(* CODESYS project NTP145_JIGA03_CPU_NX3030_0001.project
   Version: 3.61.0.0
   Project Profile: Single
   Title: Super Teste NX3030
   Company: Altus S.A.

Project tree, tasks and I/O mapping:
  Device : NX3030, Altus S.A., order no. NX3030, version 1.3.61.200
    application Application
      libraries: NX4000 Diagnostic Structs, 1.0.0.0 (WAA); NJ1001 Diagnostic Structs, 1.0.0.0 (Manufacturer); NJ1005 Diagnostic Structs, 1.0.0.1 (Manufacturer); NJ2001 Diagnostic Structs, 1.0.0.0 (Manufacturer); NJ6000 Diagnostic Structs, 1.0.0.1 (Manufacturer); NJ6001 Diagnostic Structs, 1.0.0.3 (Manufacturer); NJ6005 Diagnostic Structs, 1.0.0.9 (Manufacturer); NJ6010 Diagnostic Structs, 1.0.0.0 (Manufacturer); NJ6011 Diagnostic Structs, 1.0.0.0 (Manufacturer); NJ6020 Diagnostic Structs, 1.0.0.3 (Manufacturer); NJ6100 Diagnostic Structs, 1.0.0.0 (Manufacturer); NJ6101 Diagnostic Structs, 1.0.0.1 (Manufacturer); LibLogs, * (Manufacturer); Util, * (System); NextoSOE, 1.0.0.1 (WAA); LibMQTT, * (Manufacturer); LibRecipeHandler, 1.0.0.2 (Manufacturer); ; RedundancyLib, 3.4.4.31 (3S - Smart Software Solutions GmbH); LibInternal, 1.0.0.15 (Manufacturer); ; NX3030 Diagnostic Structs, 1.1.2.1 (WAA); NX4010 Diagnostic Structs, 1.0.0.3 (WAA); NX5000 Diagnostic Structs, 1.0.0.5 (WAA); NX5001 Diagnostic Structs, 1.0.1.12 (WAA); NXModbus Diagnostic Structs, 1.0.0.5 (WAA); LibRtuStandard, 1.0.0.14 (Manufacturer); IEC 60870-5-104 Server Diagnostic Structs, 1.0.0.2 (Manufacturer); ; ; ; ; 
      task Configuration (cyclic, interval 9000 µs, priority 4) calls Configuration.EtherCAT_Task [Configuration.EtherCAT_Task]
      task MainTask (cyclic, interval 250 ms, priority 13, watchdog 1000 ms x 1) calls MainPrg
      task ATModbusMODBUS_Server_2 (cyclic, interval 60 ms, priority 16) calls MODBUS_Server_2_Instance.Task
      task ATModbusMODBUS_Client_2 (cyclic, interval 41 ms, priority 16) calls MODBUS_Client_2_Instance.Task
      task ATModbusMODBUS_Server_3 (cyclic, interval 20 ms, priority 16) calls MODBUS_Server_3_Instance.Task
      task ATModbusMODBUS_Client_3 (cyclic, interval 41 ms, priority 16) calls MODBUS_Client_3_Instance.Task
      task ATModbusMODBUS_Slave_1 (cyclic, interval 60 ms, priority 16) calls MODBUS_Slave_1_Instance.Task
      task ATModbusMODBUS_Master_1 (cyclic, interval 16 ms, priority 16) calls MODBUS_Master_1_Instance.Task
      Bill of Materials
      Configuration and Consumption
      SystemGVLs/
        global variables System_Diagnostics
        global variables Module_Diagnostics
        global variables IOQualities
        global variables Special_Variables_Redundant
        global variables Special_Variables
      UserGVLs/
        global variables Qualities
        global variables ReqDiagnostics
        global variables Disables
        Non-Redundant/
          global variables ATs
          global variables ProjectConstants
          global variables ModbusSymbol
          global variables NonRedData
          global variables MinMaxTimes
          global variables DiagsRetain
          global variables HwVersions
          global variables Task_Information
          global variables SymbolicsNonRedundant
          global variables NonRedPointer
        Redundant/
          global variables Languages
          global variables PIDs
          global variables QuantityOfVariables
          global variables Symbolics
          global variables Recipe
          global variables ImportExportOnline
          global variables Mask
      SystemPOUs/
        program SpecialVariablesRedundantPrg [ST]
        program SpecialVariablesPrg [ST]
        program MainPrg [ST]
      UserPOUs/
        program StartPrg [ST]
        program NonSkippedPrg [ST]
        program ActivePrg [ST]
        Redundant/
          program CheckLanguages [ST]
          program Alarms [ST]
          program CheckProfibusIOs [ST]
          program PidGenerator [ST]
          program IncrRedData [ST]
          program CheckSoe [ST]
          program StateChange [ST]
          program CheckRecipe [ST]
          program ProfibusStateChange [ST]
          program CheckNVL [ST]
          Languages/
            CFC/
              data type DUT_CFC
              function block FB_CFC [CFC]
              function block FB_CFC_2 [CFC]
              program POU_CFC_1000 [CFC]
            program POU_CFC [CFC]
            program POU_FBD [FBD]
            program POU_IL [IL]
            program POU_LD [LD]
            program POU_SFC [SFC]: Testa_LD_active, Testa_IL_active, Testa_CFC_active, Testa_SFC_active, Testa_FBD_active
          program Recursividade [ST]
          program Iec104Server [ST]: DbpCmdReceiver, StepCmdReceiver
        Non-Redundant/
          program CheckModbus4 [ST]
          program CleanStats [ST]
          program CheckRedData [ST]
          program CheckSntp [ST]
          program UserLog [ST]
          program CycleTimes [ST]
          program CheckModbus1 [ST]
          program CheckModbus3 [ST]
          program CheckModbus2 [ST]
          program CheckDiagsRetain [ST]
          program ReadHwVersions [ST]
          program CheckRam [ST]
          program CheckForcing [ST]
          program WriteHwVersionsNonActive [ST]
          program DaylightSavingTime [ST]
          program MQTT [ST]
          program CheckSpecialVariables [ST]
          program CheckSpecialVarsRed [ST]
      Symbol Configuration
      global variables PersistentVars
      UserFunctions/
        function CONCATENA_2WORD_TO_DWORD [LD]
        function iCounterIncFun [ST]
      UserFunctionsBlocks/
        function block Delay [ST]
        function block Delay1 [ST]
        function block fbTotalizador [CFC]
      UserNVLs/
        global variables NVL_Sender_BroadCast_for_all
        global variables NVL_Sender_JIGA03_Exclusive_to_JIGA01
        global variables NVL_Sender_JIGA03_Exclusive_to_JIGA02
        global variables NVL_Sender_JIGA03_Exclusive_to_JIGA05
        global variables NVL_Sender_JIGA03_Exclusive_to_JIGA07
        declarations NVL_Receiver_JIGA01_Broadcast
        declarations NVL_Receiver_JIGA01_Exclusive
        declarations NVL_Receiver_JIGA02_Broadcast
        declarations NVL_Receiver_JIGA02_Exclusive
        declarations NVL_Receiver_JIGA05_Broadcast
        declarations NVL_Receiver_JIGA05_Exclusive
        declarations NVL_Receiver_JIGA07_Broadcast
        declarations NVL_Receiver_JIGA07_Exclusive
      UserStruct/
        data type Firmware
        data type Firmware_CPU
        data type Task_Informations
        data type NVL_Result
      global variables PidRetainGVL
      program PIDControl [ST]
      RecipeManager
        recipe definition Machine01: Recipe.iRecipeValueA : INT; Recipe.iRecipeValueB : INT; Recipe.iRecipeValueC : INT
      trace Trace (task MainTask): REM05_PO2020_G0, REM05_PO1000_G0, PersistentVars.dwSlave5DigIOsErrors, Task_Information.TI_MainTask.TaskInfo.dwCurScanTime
      Redundancy Configuration
    Configuration : Bus, WAA, order no. Configuration, version 1.1.1.3
      NX3030 : NX3030, Altus S.A., order no. NX3030, version 1.3.61.200
          settings: DC sync0 cycletime = 5000; Cluster Redundancy Enable = True; Generate Error if Task Whatchdog time greater than %80 of interval time = False; Consist retain and persistent area in %Q. = False; Version of MT8500 software.Major = 3; Version of MT8500 software.Minor = 61; Version of MT8500 software.Build = 300; VFInitGenerate = True; Rack Configuration Info.Total Number of Racks = 1; Rack Configuration Info.Rack-0 Type = 9003; IOModule's Address for interrupt = 255; SNTP CONFIGURATION.IP Address of First SNTP Server = [192, 168, 16, 86]; SNTP CONFIGURATION.IP Address = [192, 168, 16, 87]; SOE VARIABLE>.BaseType = 28; SOE VARIABLE>.Address = ADR(PersistentVars.IEC_SOE_QUEUE_INFO); SOE VARIABLE>.SizeInBits = 96096; SOE VARIABLE>.TotalSizeInBits = 96096; Redundancy Without Panel. = FALSE; CurrentProjectProfileParameter = 'Single'; Enable Interface = True; Enable Interface = True
        <Empty>
        COM 1
          MODBUS_Slave_1 : MODBUS RTU Slave, WAA, version 1.0.0.11
              settings: Task Name = 'ATModbusMODBUS_Slave_1'
              unmapped channels: %QD85108 Mapping Disabling
            MODBUS_Slave_1_Mapping_000 : Coil, WAA, version 1.0.0.11
            MODBUS_Slave_1_Mapping_001 : Input Status, WAA, version 1.0.0.11
            MODBUS_Slave_1_Mapping_002 : Holding Register, WAA, version 1.0.0.11
            MODBUS_Slave_1_Mapping_003 : Input Register, WAA, version 1.0.0.11
        COM 2
          MODBUS_Master_1 : MODBUS RTU Master, WAA, version 1.0.0.12
              settings: Task Name = 'ATModbusMODBUS_Master_1'
            MODBUS_Device_11 : MODBUS Device, WAA, version 1.0.0.12
                unmapped channels: %QD85132 Mapping Disabling
              MODBUS_Device_11_Mapping_000 : Coil, WAA, version 1.0.0.12
              MODBUS_Device_11_Mapping_001 : Input Status, WAA, version 1.0.0.12
              MODBUS_Device_11_Mapping_002 : Holding Register, WAA, version 1.0.0.12
              MODBUS_Device_11_Mapping_003 : Input Register, WAA, version 1.0.0.12
              MODBUS_Device_11_Mapping_004 : Coil, WAA, version 1.0.0.12
              MODBUS_Device_11_Mapping_005 : Holding Register, WAA, version 1.0.0.12
        NET 1
            settings: IP Address = [192, 168, 23, 0]; Subnetwork Mask = [255, 255, 248, 0]; Gateway Address = [192, 168, 16, 253]; IP Address PLC A Non Active = [192, 168, 23, 1]; IP Address PLC B Non Active = [192, 168, 23, 2]; Redundant = TRUE; IP Address PLC B Active = [192, 168, 23, 0]; Enable Interface = True; Switchover in case of Ethernet failure = TRUE; Obtain an IP address automatically (Single Mode) = False
          MODBUS_Client_4 : MODBUS Symbol Client, Altus S.A., version 1.0.0.37
              settings: Diagnostic Variable.BaseType = 28; Diagnostic Variable.Address = ADR(System_Diagnostics.DG_MODBUS_Client_4); Diagnostic Variable.SizeInBits = 160; Diagnostic Variable.TotalSizeInBits = 160
            MODBUS_Device_41 : MODBUS Device, Altus S.A., version 1.0.0.37
                settings: IP Address = [192, 168, 23, 3]; Mappings definition.Count = 6; Item_00000.Value Variable.BaseType = 3; Item_00000.Value Variable.Address = ADR(ModbusSymbol.awModbus4HoldingWrite); Item_00000.Value Variable.SizeInBits = 16; Item_00000.Value Variable.TotalSizeInBits = 1920; Item_00001.Value Variable.BaseType = 3; Item_00001.Value Variable.Address = ADR(ModbusSymbol.awModbus4HoldingRead); Item_00001.Value Variable.SizeInBits = 16; Item_00001.Value Variable.TotalSizeInBits = 1920; Item_00002.Value Variable.BaseType = 0; Item_00002.Value Variable.Address = ADR(ModbusSymbol.abModbus4CoilsWrite); Item_00002.Value Variable.SizeInBits = 8; Item_00002.Value Variable.TotalSizeInBits = 15360; Item_00003.Value Variable.BaseType = 0; Item_00003.Value Variable.Address = ADR(ModbusSymbol.abModbus4CoilsRead); Item_00003.Value Variable.SizeInBits = 8; Item_00003.Value Variable.TotalSizeInBits = 15360; Item_00004.Value Variable.BaseType = 3; Item_00004.Value Variable.Address = ADR(ModbusSymbol.awModbus4InputRegRead); Item_00004.Value Variable.SizeInBits = 16; Item_00004.Value Variable.TotalSizeInBits = 1920; Item_00005.Value Variable.BaseType = 0; Item_00005.Value Variable.Address = ADR(ModbusSymbol.abModbus4StatusRead); Item_00005.Value Variable.SizeInBits = 8; Item_00005.Value Variable.TotalSizeInBits = 15360; Requests definition.Count = 6; Item_00000.Diagnostic Variable.BaseType = 28; Item_00000.Diagnostic Variable.Address = ADR(ReqDiagnostics.MODBUS_Device_41_REQDG_0001); Item_00000.Diagnostic Variable.SizeInBits = 64; Item_00000.Diagnostic Variable.TotalSizeInBits = 64; Item_00000.Disabling Variable.BaseType = 0; Item_00000.Disabling Variable.Address = ADR(Disables.MODBUS_Device_41_DISABLE_0001); Item_00000.Disabling Variable.SizeInBits = 8; Item_00000.Disabling Variable.TotalSizeInBits = 8; Item_00001.Diagnostic Variable.BaseType = 28; Item_00001.Diagnostic Variable.Address = ADR(ReqDiagnostics.MODBUS_Device_41_REQDG_0002); Item_00001.Diagnostic Variable.SizeInBits = 64; Item_00001.Diagnostic Variable.TotalSizeInBits = 64; Item_00001.Disabling Variable.BaseType = 0;
                  Item_00001.Disabling Variable.Address = ADR(Disables.MODBUS_Device_41_DISABLE_0002); Item_00001.Disabling Variable.SizeInBits = 8; Item_00001.Disabling Variable.TotalSizeInBits = 8; Item_00002.Diagnostic Variable.BaseType = 28; Item_00002.Diagnostic Variable.Address = ADR(ReqDiagnostics.MODBUS_Device_41_REQDG_0003); Item_00002.Diagnostic Variable.SizeInBits = 64; Item_00002.Diagnostic Variable.TotalSizeInBits = 64; Item_00002.Disabling Variable.BaseType = 0; Item_00002.Disabling Variable.Address = ADR(Disables.MODBUS_Device_41_DISABLE_0003); Item_00002.Disabling Variable.SizeInBits = 8; Item_00002.Disabling Variable.TotalSizeInBits = 8; Item_00003.Diagnostic Variable.BaseType = 28; Item_00003.Diagnostic Variable.Address = ADR(ReqDiagnostics.MODBUS_Device_41_REQDG_0004); Item_00003.Diagnostic Variable.SizeInBits = 64; Item_00003.Diagnostic Variable.TotalSizeInBits = 64; Item_00003.Disabling Variable.BaseType = 0; Item_00003.Disabling Variable.Address = ADR(Disables.MODBUS_Device_41_DISABLE_0004); Item_00003.Disabling Variable.SizeInBits = 8; Item_00003.Disabling Variable.TotalSizeInBits = 8; Item_00004.Diagnostic Variable.BaseType = 28; Item_00004.Diagnostic Variable.Address = ADR(ReqDiagnostics.MODBUS_Device_41_REQDG_0005); Item_00004.Diagnostic Variable.SizeInBits = 64; Item_00004.Diagnostic Variable.TotalSizeInBits = 64; Item_00004.Disabling Variable.BaseType = 0; Item_00004.Disabling Variable.Address = ADR(Disables.MODBUS_Device_41_DISABLE_0005); Item_00004.Disabling Variable.SizeInBits = 8; Item_00004.Disabling Variable.TotalSizeInBits = 8; Item_00005.Diagnostic Variable.BaseType = 28; Item_00005.Diagnostic Variable.Address = ADR(ReqDiagnostics.MODBUS_Device_41_REQDG_0006); Item_00005.Diagnostic Variable.SizeInBits = 64; Item_00005.Diagnostic Variable.TotalSizeInBits = 64; Item_00005.Disabling Variable.BaseType = 0; Item_00005.Disabling Variable.Address = ADR(Disables.MODBUS_Device_41_DISABLE_0006); Item_00005.Disabling Variable.SizeInBits = 8; Item_00005.Disabling Variable.TotalSizeInBits = 8
          MODBUS_Server_2 : MODBUS Server, WAA, version 1.0.0.13
              settings: Task Name = 'ATModbusMODBUS_Server_2'
              unmapped channels: %QD85164 Mapping Disabling
            MODBUS_Server_2_Mapping_000 : Holding Register, WAA, version 1.0.0.13
                settings: Write Filter IP = [192, 168, 23, 3]; Write Filter Mask = [255, 255, 255, 255]; Read Filter IP = [192, 168, 23, 3]; Read Filter Mask = [255, 255, 255, 255]
            MODBUS_Server_2_Mapping_001 : Coil, WAA, version 1.0.0.13
                settings: Write Filter IP = [192, 168, 23, 3]; Write Filter Mask = [255, 255, 255, 255]; Read Filter IP = [192, 168, 23, 3]; Read Filter Mask = [255, 255, 255, 255]
            MODBUS_Server_2_Mapping_002 : Input Register, WAA, version 1.0.0.13
                settings: Read Filter IP = [192, 168, 23, 3]; Read Filter Mask = [255, 255, 255, 255]
            MODBUS_Server_2_Mapping_003 : Input Status, WAA, version 1.0.0.13
                settings: Read Filter IP = [192, 168, 23, 3]; Read Filter Mask = [255, 255, 255, 255]
          IEC_104_Server : IEC 60870-5-104 Server, Altus S.A., version 1.0.0.21
              settings: Diagnostic Variable.BaseType = 28; Diagnostic Variable.Address = ADR(Module_Diagnostics.DG_IEC_104_Server); Diagnostic Variable.SizeInBits = 1472; Diagnostic Variable.TotalSizeInBits = 1472
            JIGA11_CPU_HX3040_Client : Client, Altus S.A., version 1.0.0.21
                settings: Parameter list definition.Count = 15; Item_00000.Value Variable.BaseType = 0; Item_00000.Value Variable.Address = ADR(Iec104Server.bDI); Item_00000.Value Variable.SizeInBits = 8; Item_00000.Value Variable.TotalSizeInBits = 8; Item_00001.Value Variable.BaseType = 0; Item_00001.Value Variable.Address = ADR(Iec104Server.bDO); Item_00001.Value Variable.SizeInBits = 8; Item_00001.Value Variable.TotalSizeInBits = 8; Item_00002.Value Variable.BaseType = 28; Item_00002.Value Variable.Address = ADR(Iec104Server.dbpI); Item_00002.Value Variable.SizeInBits = 16; Item_00002.Value Variable.TotalSizeInBits = 16; Item_00003.Value Variable.BaseType = 28; Item_00003.Value Variable.Address = ADR(Iec104Server.dbpO); Item_00003.Value Variable.SizeInBits = 16; Item_00003.Value Variable.TotalSizeInBits = 16; Item_00004.Value Variable.BaseType = 10; Item_00004.Value Variable.Address = ADR(Iec104Server.usiSP); Item_00004.Value Variable.SizeInBits = 8; Item_00004.Value Variable.TotalSizeInBits = 8; Item_00005.Value Variable.BaseType = 28; Item_00005.Value Variable.Address = ADR(Iec104Server.dbpStep); Item_00005.Value Variable.SizeInBits = 16; Item_00005.Value Variable.TotalSizeInBits = 16; Item_00006.Value Variable.BaseType = 7; Item_00006.Value Variable.Address = ADR(Iec104Server.iAIn); Item_00006.Value Variable.SizeInBits = 16; Item_00006.Value Variable.TotalSizeInBits = 16; Item_00007.Value Variable.BaseType = 7; Item_00007.Value Variable.Address = ADR(Iec104Server.iAOn); Item_00007.Value Variable.SizeInBits = 16; Item_00007.Value Variable.TotalSizeInBits = 16; Item_00008.Value Variable.BaseType = 7; Item_00008.Value Variable.Address = ADR(Iec104Server.iAIs); Item_00008.Value Variable.SizeInBits = 16; Item_00008.Value Variable.TotalSizeInBits = 16; Item_00009.Value Variable.BaseType = 7; Item_00009.Value Variable.Address = ADR(Iec104Server.iAOs); Item_00009.Value Variable.SizeInBits = 16;
                  Item_00009.Value Variable.TotalSizeInBits = 16; Item_00010.Value Variable.BaseType = 14; Item_00010.Value Variable.Address = ADR(Iec104Server.rAIf); Item_00010.Value Variable.SizeInBits = 32; Item_00010.Value Variable.TotalSizeInBits = 32; Item_00011.Value Variable.BaseType = 14; Item_00011.Value Variable.Address = ADR(Iec104Server.rAOf); Item_00011.Value Variable.SizeInBits = 32; Item_00011.Value Variable.TotalSizeInBits = 32; Item_00012.Value Variable.BaseType = 8; Item_00012.Value Variable.Address = ADR(Iec104Server.diIT); Item_00012.Value Variable.SizeInBits = 32; Item_00012.Value Variable.TotalSizeInBits = 32; Item_00012.Counter Variable.BaseType = 8; Item_00012.Counter Variable.Address = ADR(IEC104Server.diITCounter); Item_00012.Counter Variable.SizeInBits = 32; Item_00012.Counter Variable.TotalSizeInBits = 32; Item_00013.Value Variable.BaseType = 10; Item_00013.Value Variable.Address = ADR(Iec104Server.usiJigId); Item_00013.Value Variable.SizeInBits = 8; Item_00013.Value Variable.TotalSizeInBits = 8; Item_00014.Value Variable.BaseType = 10; Item_00014.Value Variable.Address = ADR(Iec104Server.usiJigId); Item_00014.Value Variable.SizeInBits = 8; Item_00014.Value Variable.TotalSizeInBits = 8
        NET 2
            settings: IP Address = [192, 168, 23, 0]; Subnetwork Mask = [255, 255, 248, 0]; IP Address PLC A Non Active = [192, 168, 23, 1]; IP Address PLC B Non Active = [192, 168, 23, 2]; IP Address PLC B Active = [192, 168, 23, 0]; Enable Interface = True; Switchover in case of Ethernet failure = TRUE
        NX8000 : NX8000, Altus S.A., order no. NX8000, version 1.3.61.200
            settings: DC sync0 cycletime = 5000; Diag Instance Id = 0
        NX4010 : NX4010, Altus S.A., order no. NX4010, version 1.3.61.200
            settings: Physical Address of the Slave = 4; DC sync0 cycletime = 5000; Diag Instance Id = 4; %Q Start Address of Diagnostics Area = 82634; Input Offset = 81920; Output Offset = 81920
            unmapped channels: %QB81920 Reserved, %IW81920 Reserved
        NX5001_2 : NX5001, Altus S.A., order no. NX5001, version 1.1.1.19
            settings: Physical Address of the Slave = 8; Diag Instance Id = 8; %Q Start Address of Module Diagnostics Area = 83000; %Q Start Address of Slaves Diagnostics Area = 65536; User Commands Offset = 81921; NX5001R = 1; Fast Diagnostics Offset = 81924; DpParameter.Station address = 1; UseDefaults = FALSE
            unmapped channels: %QB81921 User Commands, %IW81924 User Status
        NX5001_3 : NX5001, Altus S.A., order no. NX5001, version 1.1.1.19
            settings: Physical Address of the Slave = 16; Diag Instance Id = 16; %Q Start Address of Module Diagnostics Area = 83086; %Q Start Address of Slaves Diagnostics Area = 65717; User Commands Offset = 81923; Identification = 2; Fast Diagnostics Offset = 81928; Manual user change the %Q Start Address of Slaves = TRUE; SlaveMaxDiagDataLen.Slave0 = 25; DpParameter.Station address = 1
            unmapped channels: %QB81923 User Commands, %IW81928 User Status
          PO5063_04 : PO5063, Altus S.A., order no. PO5063, version Revision=1.30, HW=V100, SW=5.00
              settings: SlavePrmData.wdFact1 = 1; SlavePrmData.wdFact2 = 100; SlavePrmData.userPrmData.userParameter = [0,4,35,0,20]; StationAddress = 4
            REM04_PO1000 : PO1000 16DI 24 Vdc Opto Coupled , Altus S.A., order no. PO1000, version Revision=1.30, HW=V100, SW=5.00
                input  REM04_PO1000_G0 : BYTE  // Input0.Byte0
                input  REM04_PO1000_G1 : BYTE  // Input0.Byte1
                unmapped channels: %IB24 Input0
        NX5000_1 : NX5000, Altus S.A., order no. NX5000, version 1.3.61.200
            settings: Physical Address of the Slave = 10; DC sync0 cycletime = 5000; Diag Instance Id = 10; %Q Start Address of Module Diagnostics Area = 83344; Network Redundancy = 1; User Commands Offset = 81929; Fast Diagnostics Offset = 81940; Enable Interface = True
            unmapped channels: %QB81929 Reserved, %IW81940 Reserved
          NET 1
              settings: IP Address = [192, 168, 23, 3]; Subnetwork Mask = [255, 255, 248, 0]; Gateway Address = [192, 168, 16, 253]; IP Address PLC A Non Active = [192, 168, 23, 4]; IP Address PLC B Non Active = [192, 168, 23, 5]; Redundant = TRUE; IP Address PLC B Active = [192, 168, 23, 3]; Enable Interface = True
            MODBUS_Server_4 : MODBUS Symbol Server, Altus S.A., version 1.0.0.8
                settings: Write Filter IP Address = [192, 168, 23, 0]; Write Filter Mask = [255, 255, 255, 248]; Read Filter IP Address = [192, 168, 23, 0]; Read Filter Mask = [255, 255, 255, 248]; Parameter list definition.Count = 4; Item_00000.Value Variable.BaseType = 3; Item_00000.Value Variable.Address = ADR(ModbusSymbol.awModbus4Holding); Item_00000.Value Variable.SizeInBits = 16; Item_00000.Value Variable.TotalSizeInBits = 1920; Item_00001.Value Variable.BaseType = 0; Item_00001.Value Variable.Address = ADR(ModbusSymbol.abModbus4Coils); Item_00001.Value Variable.SizeInBits = 8; Item_00001.Value Variable.TotalSizeInBits = 15360; Item_00002.Value Variable.BaseType = 3; Item_00002.Value Variable.Address = ADR(ModbusSymbol.awModbus4InputReg); Item_00002.Value Variable.SizeInBits = 16; Item_00002.Value Variable.TotalSizeInBits = 1920; Item_00003.Value Variable.BaseType = 0; Item_00003.Value Variable.Address = ADR(ModbusSymbol.abModbus4Status); Item_00003.Value Variable.SizeInBits = 8; Item_00003.Value Variable.TotalSizeInBits = 15360; Diagnostic Variable.BaseType = 28; Diagnostic Variable.Address = ADR(Module_Diagnostics.DG_MODBUS_Server_4); Diagnostic Variable.SizeInBits = 160; Diagnostic Variable.TotalSizeInBits = 160
            MODBUS_Client_2 : MODBUS Client, WAA, version 1.0.0.14
                settings: Task Name = 'ATModbusMODBUS_Client_2'
              MODBUS_Device_21 : MODBUS Device, WAA, version 1.0.0.14
                  settings: Destination IP = [192, 168, 23, 0]
                  unmapped channels: %QD85020 Mapping Disabling
                MODBUS_Device_21_Mapping_001 : Holding Register, WAA, version 1.0.0.14
                MODBUS_Device_21_Mapping_002 : Holding Register, WAA, version 1.0.0.14
                MODBUS_Device_21_Mapping_003 : Coil, WAA, version 1.0.0.14
                MODBUS_Device_21_Mapping_004 : Coil, WAA, version 1.0.0.14
                MODBUS_Device_21_Mapping_005 : Input Register, WAA, version 1.0.0.14
                MODBUS_Device_21_Mapping_006 : Input Status, WAA, version 1.0.0.14
            MODBUS_Server_3 : MODBUS Server, WAA, version 1.0.0.13
                settings: Task Name = 'ATModbusMODBUS_Server_3'
                unmapped channels: %QD85052 Mapping Disabling
              MODBUS_Server_3_Mapping_001 : Holding Register, WAA, version 1.0.0.13
                  settings: Write Filter IP = [192, 168, 23, 6]; Write Filter Mask = [255, 255, 255, 255]; Read Filter IP = [192, 168, 23, 6]; Read Filter Mask = [255, 255, 255, 255]
              MODBUS_Server_3_Mapping_002 : Coil, WAA, version 1.0.0.13
                  settings: Write Filter IP = [192, 168, 23, 6]; Write Filter Mask = [255, 255, 255, 255]; Read Filter IP = [192, 168, 23, 6]; Read Filter Mask = [255, 255, 255, 255]
              MODBUS_Server_3_Mapping_003 : Input Register, WAA, version 1.0.0.13
                  settings: Read Filter IP = [192, 168, 23, 6]; Read Filter Mask = [255, 255, 255, 255]
              MODBUS_Server_3_Mapping_004 : Input Status, WAA, version 1.0.0.13
                  settings: Read Filter IP = [192, 168, 23, 6]; Read Filter Mask = [255, 255, 255, 255]
        NX5000_2 : NX5000, Altus S.A., order no. NX5000, version 1.3.61.200
            settings: Physical Address of the Slave = 12; DC sync0 cycletime = 5000; Diag Instance Id = 12; %Q Start Address of Module Diagnostics Area = 83544; User Commands Offset = 81931; NX5000R = 1; Fast Diagnostics Offset = 81946; Enable Interface = True
            unmapped channels: %QB81931 Reserved, %IW81946 Reserved
          NET 1
              settings: IP Address = [192, 168, 23, 3]; Subnetwork Mask = [255, 255, 248, 0]; Gateway Address = [192, 168, 16, 253]; IP Address PLC A Non Active = [192, 168, 23, 4]; IP Address PLC B Non Active = [192, 168, 23, 5]; IP Address PLC B Active = [192, 168, 23, 3]; Enable Interface = True
        NX5001_1 : NX5001, Altus S.A., order no. NX5001, version 1.1.1.19
            settings: Physical Address of the Slave = 6; Diag Instance Id = 6; %Q Start Address of Module Diagnostics Area = 83172; %Q Start Address of Slaves Diagnostics Area = 65536; Network Redundancy = 1; User Commands Offset = 81925; Fast Diagnostics Offset = 81932; Manual user change the %Q Start Address of Slaves = TRUE; SlaveMaxDiagDataLen.Slave0 = 25; SlaveMaxDiagDataLen.Slave1 = 25; DpParameter.Station address = 1; UseDefaults = FALSE
            unmapped channels: %QB81925 User Commands, %IW81932 User Status
          PO5065_05 : PO5065, Altus S.A., order no. PO5065, version Revision=1.30, HW=V100, SW=1.01
              settings: SlavePrmData.wdFact1 = 1; SlavePrmData.wdFact2 = 100; SlavePrmData.userPrmData.userParameter = [0, 0, 0, 0, 4, 98, 0, 20]; StationAddress = 5
            REM05_PO1000 : PO1000 16DI 24 Vdc Opto Coupled , Altus S.A., order no. PO1000, version Revision=1.30, HW=V100, SW=1.01
                input  REM05_PO1000_G0 : BYTE  // Input0.Byte0
                input  REM05_PO1000_G1 : BYTE  // Input0.Byte1
                unmapped channels: %IB0 Input0
            REM05_PO2020 : PO2020 16DO Transistor Opto     , Altus S.A., order no. PO2020, version Revision=1.30, HW=V100, SW=1.01
                output REM05_PO2020_G0 : BYTE  // Output0.Byte0
                output REM05_PO2020_G1 : BYTE  // Output0.Byte1
                unmapped channels: %QB2000 Output0
            REM05_PO9100 : PO9100 - Redundant Head PO5065  , Altus S.A., order no. PO9100_RH, version Revision=1.30, HW=V100, SW=1.01
                input  REM05_PO5065_IN AT %IW2 : WORD  // Input0
                output REM05_PO5065_OUT AT %QW2002 : WORD  // Output0
          PO5065_10 : PO5065, Altus S.A., order no. PO5065, version Revision=1.30, HW=V100, SW=1.01
              settings: SlavePrmData.wdFact1 = 1; SlavePrmData.wdFact2 = 100; SlavePrmData.userPrmData.userParameter = [0, 0, 0, 0, 4, 98, 0, 20]; StationAddress = 10
            REM10_PO1212 : PO1212 8AI Universal Isolated   , Altus S.A., order no. PO1212, version Revision=1.30, HW=V100, SW=1.01
                settings: ExtPrmData.userParameter = [10, 8, 10, 4, 4, 4, 4, 4, 4, 4]
                input  REM10_PO1212_C00 : WORD  // Input0.Word0
                input  REM10_PO1212_C01 : WORD  // Input0.Word1
                input  REM10_PO1212_C02 : WORD  // Input0.Word2
                input  REM10_PO1212_C03 : WORD  // Input0.Word3
                input  REM10_PO1212_C04 : WORD  // Input0.Word4
                input  REM10_PO1212_C05 : WORD  // Input0.Word5
                input  REM10_PO1212_C06 : WORD  // Input0.Word6
                input  REM10_PO1212_C07 : WORD  // Input0.Word7
                unmapped channels: %IW4 Input0
            REM10_PO2132 : PO2132 4AO Universal Isolated   , Altus S.A., order no. PO2132, version Revision=1.30, HW=V100, SW=1.01
                settings: ExtPrmData.userParameter = [6, 0, 0, 2, 2, 2]
                output REM10_PO2132_C00 : WORD  // Output0.Word0
                output REM10_PO2132_C01 : WORD  // Output0.Word1
                output REM10_PO2132_C02 : WORD  // Output0.Word2
                output REM10_PO2132_C03 : WORD  // Output0.Word3
                unmapped channels: %QW2004 Output0
            REM10_PO9100 : PO9100 - Redundant Head PO5065  , Altus S.A., order no. PO9100_RH, version Revision=1.30, HW=V100, SW=1.01
                input  REM10_PO5065_IN AT %IW20 : WORD  // Input0
                output REM10_PO5065_OUT AT %QW2012 : WORD  // Output0
        NX5000_3 : NX5000, Altus S.A., order no. NX5000, version 1.3.61.200
            settings: Physical Address of the Slave = 20; DC sync0 cycletime = 5000; Diag Instance Id = 20; %Q Start Address of Module Diagnostics Area = 83744; User Commands Offset = 81933; Fast Diagnostics Offset = 81952; Enable Interface = True
            unmapped channels: %QB81933 Reserved, %IW81952 Reserved
          NET 1
              settings: IP Address = [192, 168, 23, 6]; Subnetwork Mask = [255, 255, 248, 0]; Gateway Address = [192, 168, 16, 253]; IP Address PLC A Non Active = [192, 168, 23, 7]; IP Address PLC B Non Active = [192, 168, 23, 8]; IP Address PLC B Active = [192, 168, 23, 6]; Enable Interface = True
            MODBUS_Client_3 : MODBUS Client, WAA, version 1.0.0.14
                settings: Task Name = 'ATModbusMODBUS_Client_3'
              MODBUS_Device_31 : MODBUS Device, WAA, version 1.0.0.14
                  settings: Destination IP = [192, 168, 23, 3]
                  unmapped channels: %QD85076 Mapping Disabling
                MODBUS_Device_31_Mapping_000 : Holding Register, WAA, version 1.0.0.14
                MODBUS_Device_31_Mapping_001 : Holding Register, WAA, version 1.0.0.14
                MODBUS_Device_31_Mapping_002 : Coil, WAA, version 1.0.0.14
                MODBUS_Device_31_Mapping_003 : Coil, WAA, version 1.0.0.14
                MODBUS_Device_31_Mapping_004 : Input Register, WAA, version 1.0.0.14
                MODBUS_Device_31_Mapping_005 : Input Status, WAA, version 1.0.0.14
  Library Information/
    function GetLibVersion [ST]
    function GetLibVersionNumber [ST]
    function IsLibReleased [ST]
  Project Information/
    function GetCompany [ST]
    function GetTitle [ST]
    function GetVersion [ST]
    function GetTextProperty [ST]
    function GetTextProperty2 [ST]
    function GetNumberProperty [ST]
    function GetBooleanProperty [ST]
    function GetVersionProperty [ST]
  function ForceScanTime [ST]
*)

// Device/Application/UserPOUs/Redundant/Languages/CFC/DUT_CFC
TYPE DUT_CFC :
STRUCT
	iVar01_Add_A: INT;
	iVar02_Add_B: INT;
END_STRUCT
END_TYPE

// Device/Application/UserStruct/Firmware
TYPE Firmware :
STRUCT
	dwFirmwareVersion:	DWORD; // Versão Firmware do produto em Hexadecimal
	uiSlaveAddress: 	UINT; // Rack e Slot do produto em Hexadecimal
	dwProductID:		DWORD; // Modelo do produto em Hexadecimal
	iIndex:				INT; // Ponteiro do local das informações lidas do NextoBus.
END_STRUCT
END_TYPE

// Device/Application/UserStruct/Firmware_CPU
TYPE Firmware_CPU :
STRUCT
	abyCPUVersion: ARRAY[0..3] OF BYTE;		   // Versão da CPU
	abyBootloaderVersion: ARRAY[0..3] OF BYTE; // Versão da CPU
	abyProcAuxVersion: ARRAY[0..3] OF BYTE;	   // Versão da CPU
	dwCPUModel: DWORD;                         // Modelo da CPU
END_STRUCT
END_TYPE

// Device/Application/UserStruct/Task_Informations
TYPE Task_Informations :
STRUCT
	sTaskName:			STRING;						// Variável recebe o nome da tarefa.
	psTaskName:			POINTER TO STRING;			// Ponteiro com o nome da tarefa.
	pstTaskInfo:		POINTER TO stTaskInfo;		// Ponteiro que irá receber as informações da tarefa.
	TaskInfo:			stTaskInfo;					// Retona aqui as Informações sobre a tarefa
END_STRUCT
END_TYPE

// Device/Application/UserStruct/NVL_Result
TYPE NVL_Result :
STRUCT
	iTempoMinimo 				:	INT;	// Tempo do menor intervalo de comunicação
	iTempoMedio					:	INT;	// Tempo médio de intervalo de comunicação
	iTempoMaximo				:	INT;	// Tempo do maior intervalo de comunicação (limite 30000)
	lwQtdTotalComunicacoes		:	LWORD;	// Quantidade total de comunicações realizadas
	wQtdComMaior3segundos		: 	WORD;	//Quantidde de comunicações acima de 3 segundos
	wQtdComMaior4segundos		: 	WORD;	//Quantidde de comunicações acima de 3 segundos
	wQtdComMaior5segundos		: 	WORD;	//Quantidde de comunicações acima de 3 segundos
END_STRUCT
END_TYPE

// Device/Application/SystemGVLs/System_Diagnostics
VAR_GLOBAL
	//DG_MODBUS_Client_4 diagnostics variable
	DG_MODBUS_Client_4                          : T_DIAG_MODBUS_ETH_CLIENT_1;
	//DG_PO5065_05 diagnostics variable
	DG_PO5065_05                    AT %QB65536 : T_DIAG_PO5065_1;
	//DG_REM05_PO1000 diagnostics variable
	DG_REM05_PO1000                 AT %QB65561 : T_DIAG_PO1000_1;
	//DG_REM05_PO2020 diagnostics variable
	DG_REM05_PO2020                 AT %QB65571 : T_DIAG_PO2020_1;
	//DG_REM05_PO9100 diagnostics variable
	DG_REM05_PO9100                 AT %QB65581 : T_DIAG_VIRTUAL_MODULE_1;
	//DG_PO5065_10 diagnostics variable
	DG_PO5065_10                    AT %QB65591 : T_DIAG_PO5065_1;
	//DG_REM10_PO1212 diagnostics variable
	DG_REM10_PO1212                 AT %QB65616 : T_DIAG_PO1212_1;
	//DG_REM10_PO2132 diagnostics variable
	DG_REM10_PO2132                 AT %QB65626 : T_DIAG_PO2134_1;
	//DG_REM10_PO9100 diagnostics variable
	DG_REM10_PO9100                 AT %QB65636 : T_DIAG_VIRTUAL_MODULE_1;
	//DG_PO5063_04 diagnostics variable
	DG_PO5063_04                    AT %QB65717 : T_DIAG_PO5063_1;
	//DG_REM04_PO1000 diagnostics variable
	DG_REM04_PO1000                 AT %QB65742 : T_DIAG_PO1000_1;
	//DG_NX3030 diagnostics variable
	DG_NX3030                       AT %QB81941 : T_DIAG_NX3030_1;
	//DG_MODBUS_Client_2 diagnostics variable
	DG_MODBUS_Client_2              AT %QB85000 : T_DIAG_MODBUS_ETH_CLIENT_1;
	//DG_MODBUS_Device_21_Mapping_001 diagnostics variable
	DG_MODBUS_Device_21_Mapping_001 AT %QB85024 : T_DIAG_MODBUS_ETH_MAPPING_1;
	//DG_MODBUS_Client_3 diagnostics variable
	DG_MODBUS_Client_3              AT %QB85056 : T_DIAG_MODBUS_ETH_CLIENT_1;
	//DG_MODBUS_Device_31_Mapping_000 diagnostics variable
	DG_MODBUS_Device_31_Mapping_000 AT %QB85080 : T_DIAG_MODBUS_ETH_MAPPING_1;
	//DG_MODBUS_Master_1 diagnostics variable
	DG_MODBUS_Master_1              AT %QB85112 : T_DIAG_MODBUS_RTU_MASTER_1;
	//DG_MODBUS_Device_11_Mapping_000 diagnostics variable
	DG_MODBUS_Device_11_Mapping_000 AT %QB85136 : T_DIAG_MODBUS_RTU_MAPPING_1;
	//DG_MODBUS_Device_11_Mapping_001 diagnostics variable
	DG_MODBUS_Device_11_Mapping_001 AT %QB85168 : T_DIAG_MODBUS_RTU_MAPPING_1;
	//DG_MODBUS_Device_11_Mapping_002 diagnostics variable
	DG_MODBUS_Device_11_Mapping_002 AT %QB85176 : T_DIAG_MODBUS_RTU_MAPPING_1;
	//DG_MODBUS_Device_11_Mapping_003 diagnostics variable
	DG_MODBUS_Device_11_Mapping_003 AT %QB85184 : T_DIAG_MODBUS_RTU_MAPPING_1;
	//DG_MODBUS_Device_11_Mapping_004 diagnostics variable
	DG_MODBUS_Device_11_Mapping_004 AT %QB85192 : T_DIAG_MODBUS_RTU_MAPPING_1;
	//DG_MODBUS_Device_11_Mapping_005 diagnostics variable
	DG_MODBUS_Device_11_Mapping_005 AT %QB85200 : T_DIAG_MODBUS_RTU_MAPPING_1;
	//DG_MODBUS_Device_31_Mapping_001 diagnostics variable
	DG_MODBUS_Device_31_Mapping_001 AT %QB85208 : T_DIAG_MODBUS_ETH_MAPPING_1;
	//DG_MODBUS_Device_31_Mapping_002 diagnostics variable
	DG_MODBUS_Device_31_Mapping_002 AT %QB85216 : T_DIAG_MODBUS_ETH_MAPPING_1;
	//DG_MODBUS_Device_31_Mapping_003 diagnostics variable
	DG_MODBUS_Device_31_Mapping_003 AT %QB85224 : T_DIAG_MODBUS_ETH_MAPPING_1;
	//DG_MODBUS_Device_31_Mapping_004 diagnostics variable
	DG_MODBUS_Device_31_Mapping_004 AT %QB85232 : T_DIAG_MODBUS_ETH_MAPPING_1;
	//DG_MODBUS_Device_31_Mapping_005 diagnostics variable
	DG_MODBUS_Device_31_Mapping_005 AT %QB85240 : T_DIAG_MODBUS_ETH_MAPPING_1;
	//DG_MODBUS_Device_21_Mapping_002 diagnostics variable
	DG_MODBUS_Device_21_Mapping_002 AT %QB85248 : T_DIAG_MODBUS_ETH_MAPPING_1;
	//DG_MODBUS_Device_21_Mapping_003 diagnostics variable
	DG_MODBUS_Device_21_Mapping_003 AT %QB85256 : T_DIAG_MODBUS_ETH_MAPPING_1;
	//DG_MODBUS_Device_21_Mapping_004 diagnostics variable
	DG_MODBUS_Device_21_Mapping_004 AT %QB85264 : T_DIAG_MODBUS_ETH_MAPPING_1;
	//DG_MODBUS_Device_21_Mapping_005 diagnostics variable
	DG_MODBUS_Device_21_Mapping_005 AT %QB85272 : T_DIAG_MODBUS_ETH_MAPPING_1;
	//DG_MODBUS_Device_21_Mapping_006 diagnostics variable
	DG_MODBUS_Device_21_Mapping_006 AT %QB85280 : T_DIAG_MODBUS_ETH_MAPPING_1;
END_VAR

// Device/Application/SystemGVLs/Module_Diagnostics
VAR_GLOBAL
	//DG_IEC_104_Server diagnostics variable
	DG_IEC_104_Server              : T_DIAG_IEC104_SERVER_1;
	//DG_MODBUS_Server_4 diagnostics variable
	DG_MODBUS_Server_4             : T_DIAG_MODBUS_ETH_SERVER_1;
	//DG_NX4010 diagnostics variable
	DG_NX4010          AT %QB82634 : T_DIAG_NX4010_1;
	//DG_NX5001_2 diagnostics variable
	DG_NX5001_2        AT %QB83000 : T_DIAG_NX5001_1;
	//DG_NX5001_3 diagnostics variable
	DG_NX5001_3        AT %QB83086 : T_DIAG_NX5001_1;
	//DG_NX5001_1 diagnostics variable
	DG_NX5001_1        AT %QB83172 : T_DIAG_NX5001_1;
	//DG_NX5000_1 diagnostics variable
	DG_NX5000_1        AT %QB83344 : T_DIAG_NX5000_1;
	//DG_NX5000_2 diagnostics variable
	DG_NX5000_2        AT %QB83544 : T_DIAG_NX5000_1;
	//DG_NX5000_3 diagnostics variable
	DG_NX5000_3        AT %QB83744 : T_DIAG_NX5000_1;
	//DG_MODBUS_Server_3 diagnostics variable
	DG_MODBUS_Server_3 AT %QB85032 : T_DIAG_MODBUS_ETH_SERVER_1;
	//DG_MODBUS_Slave_1 diagnostics variable
	DG_MODBUS_Slave_1  AT %QB85088 : T_DIAG_MODBUS_RTU_SLAVE_1;
	//DG_MODBUS_Server_2 diagnostics variable
	DG_MODBUS_Server_2 AT %QB85144 : T_DIAG_MODBUS_ETH_SERVER_1;
END_VAR

// Device/Application/UserGVLs/Qualities
VAR_GLOBAL
END_VAR

// Device/Application/UserGVLs/ReqDiagnostics
VAR_GLOBAL
	MODBUS_Device_41_REQDG_0001 : NXMODBUS_DIAGNOSTIC_STRUCTS.T_DIAG_MODBUS_ETH_MAPPING_1;
	MODBUS_Device_41_REQDG_0002 : NXMODBUS_DIAGNOSTIC_STRUCTS.T_DIAG_MODBUS_ETH_MAPPING_1;
	MODBUS_Device_41_REQDG_0003 : NXMODBUS_DIAGNOSTIC_STRUCTS.T_DIAG_MODBUS_ETH_MAPPING_1;
	MODBUS_Device_41_REQDG_0004 : NXMODBUS_DIAGNOSTIC_STRUCTS.T_DIAG_MODBUS_ETH_MAPPING_1;
	MODBUS_Device_41_REQDG_0005 : NXMODBUS_DIAGNOSTIC_STRUCTS.T_DIAG_MODBUS_ETH_MAPPING_1;
	MODBUS_Device_41_REQDG_0006 : NXMODBUS_DIAGNOSTIC_STRUCTS.T_DIAG_MODBUS_ETH_MAPPING_1;
END_VAR

// Device/Application/UserGVLs/Disables
VAR_GLOBAL
	MODBUS_Device_41_DISABLE_0001: BOOL;
	MODBUS_Device_41_DISABLE_0002: BOOL;
	MODBUS_Device_41_DISABLE_0003: BOOL;
	MODBUS_Device_41_DISABLE_0004: BOOL;
	MODBUS_Device_41_DISABLE_0005: BOOL;
	MODBUS_Device_41_DISABLE_0006: BOOL;
END_VAR

// Device/Application/SystemGVLs/IOQualities
VAR_GLOBAL
END_VAR

// Device/Application/SystemGVLs/Special_Variables_Redundant
(*This GVL is blocked to edit.*)
VAR_GLOBAL
	Pulse_100ms_Redundant      : BOOL;                     //Pulse signal with 100ms period (toggles every 50ms)
	Pulse_500ms_Redundant      : BOOL;                     //Pulse signal with 500ms period (toggles every 250ms)
	Pulse_1s_Redundant         : BOOL;                     //Pulse signal with 1s period (toggles every 500ms)
	Pulse_2s_Redundant         : BOOL;                     //Pulse signal with 2s period (toggles every 1s)
	Pulse_5s_Redundant         : BOOL;                     //Pulse signal with 5s period (toggles every 2,5s)
	Pulse_10s_Redundant        : BOOL;                     //Pulse signal with 10s period (toggles every 5s)
	Pulse_30s_Redundant        : BOOL;                     //Pulse signal with 30s period (toggles every 15s)
	Pulse_60s_Redundant        : BOOL;                     //Pulse signal with 60s period (toggles every 30s)
	Pulse_Scan_Redundant       : BOOL;                     //Scan pulse that toggles every MainTask cycle
END_VAR

// Device/Application/SystemGVLs/Special_Variables
(*This GVL is blocked to edit.*)
VAR_GLOBAL
	Pulse_100ms : BOOL;                     //Pulse signal with 100ms period (toggles every 50ms)
	Pulse_500ms : BOOL;                     //Pulse signal with 500ms period (toggles every 250ms)
	Pulse_1s    : BOOL;                     //Pulse signal with 1s period (toggles every 500ms)
	Pulse_2s    : BOOL;                     //Pulse signal with 2s period (toggles every 1s)
	Pulse_5s    : BOOL;                     //Pulse signal with 5s period (toggles every 2,5s)
	Pulse_10s   : BOOL;                     //Pulse signal with 10s period (toggles every 5s)
	Pulse_30s   : BOOL;                     //Pulse signal with 30s period (toggles every 15s)
	Pulse_60s   : BOOL;                     //Pulse signal with 60s period (toggles every 30s)
	Pulse_Scan  : BOOL;                     //Scan pulse that toggles every MainTask cycle
	System_Time : EXTENDED_DATE_AND_TIME;   //System date and time
	Day_Of_Week : DAYS_OF_WEEK;             //Day of week
	Hour_Minute : UINT;                     //Integer variable with hour and minute (hour*100 + minute)
END_VAR

VAR_GLOBAL CONSTANT
	udiMainTaskInterval : UDINT := 250000;     //MainTask configured interval [us].
END_VAR

// Device/Application/PersistentVars
// Gerenciamento e Resumo dos testes
//{attribute 'qualified_only'} // BUG 21281
{attribute 'symbol' := 'none'} 
VAR_GLOBAL PERSISTENT RETAIN // RESULTADOS DOS TESTES
	iBug17184_Counter_MDBUS3:			INT;			// Contador de vezes que o bug 17184 ocorreu no MODBUS 3.
	iBug17184_Counter_MDBUS4:			INT;			// Contador de vezes que o bug 17184 ocorreu no MODBUS 4.
	iBug17184_CounterDig_MDBUS3:		INT;			// Contador de vezes que o bug 17184 ocorreu no MODBUS 3.
	iBug17184_CounterDig_MDBUS4:		INT;			// Contador de vezes que o bug 17184 ocorreu no MODBUS 4.
	{attribute 'symbol' := 'readwrite'}
	bStartTest:							BOOL:= FALSE;	// Habilita a execução do super teste
	{attribute 'symbol' := 'readwrite'}
	bEnableCleanStats:					BOOL:= TRUE;	// Apaga as estatísticas em PersistentVars
	{attribute 'symbol' := 'readwrite'}
	bEnableStateChange:					BOOL:= TRUE;	// Habilita a troca de estados automática
	{attribute 'symbol' := 'read'}
 	bCheckForcingBoolVar:    			BOOL:= FALSE;	// Forçar para TRUE antes de habilitar o super-teste
	{attribute 'symbol' := 'read'}
	bCheckForcingWordVar:   			WORD:= 0;		// Forçar para 12345 antes de habilitar o super-teste
	{attribute 'symbol' := 'read'}
	tElapsedTimeToFailure:				TIME;			// Tempo de teste até ocorrência da falha
	{attribute 'symbol' := 'read'}
	byCurRedStatePlcA:					REDUNDANCY_STATE;	// Estado de redundância atual do PLC A
	{attribute 'symbol' := 'read'}
	byCurRedStatePlcB:					REDUNDANCY_STATE;	// Estado de redundância atual do PLC B
	{attribute 'symbol' := 'read'}
	bFailureDetected:					BOOL;			// Algum dos testes detectou uma falha, ver abaixo
		{attribute 'symbol' := 'read'}
		bActiveDiagPlcA:				BOOL;			// Houve algum diagnóstico ativo indevido no PLC A
		{attribute 'symbol' := 'read'}
		bActiveDiagPlcB:				BOOL;			// Houve algum diagnóstico ativo indevido no PLC B
		{attribute 'symbol' := 'read'}
		bLanguages:						BOOL;			// Houve falha no teste das linguagens de programação
		{attribute 'symbol' := 'read'}
		bModbus1:						BOOL;			// Houve falha no teste de consistências dos dados trocados pelo MODBUS 1
		{attribute 'symbol' := 'read'}	
		bModbus2:						BOOL;			// Houve falha no teste de consistências dos dados trocados pelo MODBUS 2
		{attribute 'symbol' := 'read'}	
		bModbus3:						BOOL;			// Houve falha no teste de consistências dos dados trocados pelo MODBUS 3
		{attribute 'symbol' := 'read'}	
		bModbus4:						BOOL;			// Houve falha no teste de consistências dos dados trocados pelo MODBUS 4
		{attribute 'symbol' := 'read'}
		bIec104:						BOOL;			// Não implementado
		{attribute 'symbol' := 'read'}
		bProfibusIOs:					BOOL;			// Houve falha no teste de consistência de E/S Profibus
		{attribute 'symbol' := 'read'}
		bRecipeManager:					BOOL;			// Houve falha no teste de consistência do Recipe Manager
		{attribute 'symbol' := 'read'}
		bRedundantData:					BOOL;			// Houve falha no teste de sincronização de dados redundantes
		{attribute 'symbol' := 'read'}
		bRedundantState:				BOOL;			// Houve falha no teste de troca de estados de redundância
		{attribute 'symbol' := 'read'}
		bSNTP:							BOOL;			// Houve falha no teste de SNTP
		{attribute 'symbol' := 'read'}
		bSOE:							BOOL;			// Houve falha no teste de SOE
		{attribute 'symbol' := 'read'}
		bUserLog:						BOOL;			// Houve falha no teste da função Userlog
		{attribute 'symbol' := 'read'}
		bRam:							BOOL;			// Houve falha no teste de consistências da memória RAM da UCP
		{attribute 'symbol' := 'read'}
		bForcing:						BOOL;			// Houve falha no teste de consistências da memória Forçamentos da UCP
		{attribute 'symbol' := 'read'}
		bSpecialVariables:				BOOL;			// Houve falha no teste de consistências das variáveis especiais
	// Resultados da POU CycleTimes:
	{attribute 'symbol' := 'read'}	
	dwPLCAMainTaskCurScanTime:			DWORD;	// Tempo de ciclo corrente da tarefa MainTask PLCA
	{attribute 'symbol' := 'read'}
	dwPLCAMainTaskMaxScanTime: 		 	DWORD;	// Tempo de ciclo máximo da tarefa MainTask PLCA
	{attribute 'symbol' := 'read'}
	dwPLCAMainTaskAvgScanTime: 		 	DWORD;	// Tempo de ciclo médio da tarefa MainTask PLCA
	{attribute 'symbol' := 'read'}
	dwPLCAMainTaskMinScanTime: 		 	DWORD;	// Tempo de ciclo mínimo da tarefa MainTask PLCA
	dwPLCAConfigurationCurScanTime:		DWORD;	// Tempo de ciclo corrente da tarefa Configuration PLCA
	dwPLCAConfigurationMaxScanTime:		DWORD;	// Tempo de ciclo máximo da tarefa Configuration PLCA
	dwPLCAConfigurationAvgScanTime:		DWORD;	// Tempo de ciclo médio da tarefa Configuration PLCA
	dwPLCAConfigurationMinScanTime:		DWORD;	// Tempo de ciclo mínimo da tarefa Configuration PLCA
	{attribute 'symbol' := 'read'}	
	dwPLCBMainTaskCurScanTime:			DWORD;	// Tempo de ciclo corrente da tarefa MainTask PLCB
	{attribute 'symbol' := 'read'}
	dwPLCBMainTaskMaxScanTime: 		 	DWORD;	// Tempo de ciclo máximo da tarefa MainTask PLCB
	{attribute 'symbol' := 'read'}
	dwPLCBMainTaskAvgScanTime: 		 	DWORD;	// Tempo de ciclo médio da tarefa MainTask PLCB
	{attribute 'symbol' := 'read'}
	dwPLCBMainTaskMinScanTime: 		 	DWORD;	// Tempo de ciclo mínimo da tarefa MainTask PLCB
	dwPLCBConfigurationCurScanTime:		DWORD;	// Tempo de ciclo corrente da tarefa Configuration PLCB
	dwPLCBConfigurationMaxScanTime:		DWORD;	// Tempo de ciclo máximo da tarefa Configuration PLCB
	dwPLCBConfigurationAvgScanTime:		DWORD;	// Tempo de ciclo médio da tarefa Configuration PLCB
	dwPLCBConfigurationMinScanTime:		DWORD;	// Tempo de ciclo mínimo da tarefa Configuration PLCB
	{attribute 'symbol' := 'read'}
	dwPLCAMainTaskLoadMax: 				DWORD:= 0;	// Percentual máximo de consumo da MainTask PLCA
	{attribute 'symbol' := 'read'}
	dwPLCAMainTaskLoadAvg: 				DWORD;	// Percentual instantâneo de consumo da MainTask PLCA
	{attribute 'symbol' := 'read'}
	dwPLCAMainTaskLoadMin: 				DWORD:= 10000;	// Percentual mínimo de consumo da MainTask PLCA
	{attribute 'symbol' := 'read'}
	dwPLCBMainTaskLoadMax: 				DWORD:= 0;	// Percentual máximo de consumo da MainTask PLCB
	{attribute 'symbol' := 'read'}
	dwPLCBMainTaskLoadAvg: 				DWORD;	// Percentual instantâneo de consumo da MainTask PLCB
	{attribute 'symbol' := 'read'}
	dwPLCBMainTaskLoadMin: 				DWORD:= 10000;	// Percentual mínimo de consumo da MainTask PLCB
	// Resultados da POU CheckRam:
	{attribute 'symbol' := 'read'}
	dwMinFreeRamPlcA:					DWORD;			// Memória livre mínima PLCA
	{attribute 'symbol' := 'read'}
	dwMaxFreeRamPlcA:					DWORD;			// Memória livre máxima PLCA
	{attribute 'symbol' := 'read'}
	dwMinFreeRamPlcB:					DWORD;			// Memória livre mínima PLCB
	{attribute 'symbol' := 'read'}
	dwMaxFreeRamPlcB:					DWORD;			// Memória livre máxima PLCB
	{attribute 'symbol' := 'read'}
	dwInstFreeRamPlcA:						DWORD;			// Memória livre instantânea PLCA
	{attribute 'symbol' := 'read'}
	dwInstFreeRamPlcB:						DWORD;			// Memória livre instantânea PLCB		
	bRamTotalFailure:					BOOL;
	bRamFreeVarFailure:					BOOL;
	// Resultados da POU StateChange:
	bExchangeStateFail: 			 	BOOL; 	// Houve falha na troca de estados
	dwTransitionsCnt: 				 	DWORD; 	// Contador de transições de estado
	dwSwitchoverCnt:				 	DWORD;	// Contador de switchovers
	// Resultados da POU ProfibusStateChange:
	dwPBSwitchoverCnt:				 	DWORD;	// Contador de switchovers remota Profibus 99
	// Resultados da POU SNTP_PLCx:
	bSntpServerFailures:				BOOL;
	bSntpSourceFailures:				BOOL;
	bTimezoneFailure:					BOOL;
	iSntpSyncFailures:					INT;
	// Resultados da POU CheckSoe:
	bSOE1EventsMismatch: 			 	BOOL;	// A quantidade de eventos registrados no Servidor SOE 1 é diferente da quantidade de eventos gerados
	bSOE1FalseOverflow:					BOOL;	// O diagnóstico de overflow do Cliente SOE 1 foi acionado sem que o limite de eventos tenha sido gerado
	bSOE2EventsMismatch:				BOOL;	// A quantidade de eventos registrados no Servidor SOE 2 é diferente da quantidade de eventos gerados
	bSOE2FalseOverflow:					BOOL;	// O diagnóstico de overflow do Cliente SOE 2 foi acionado sem que o limite de eventos tenha sido gerado
	// Resultados das POUs CheckRedData e IncrRedData:
	iSyncFailCntSymb: 			 		INT;	// Contador de falhas de sincronização de variáveis simbólicas
	iSyncFailCntQ:						INT;	// Contador de falhas de sincronização de %Q
	iSyncFailCntM:						INT;	// Contador de falhas de sincronização de %M 
	iSyncFailCntI:						INT;	// Contador de falhas de sincronização de %I
	iSyncFailCallback_vfInit:			INT;	// Contador de falhas da rotina de Callback_vfInit necessária para sincronizar os ponteiros de Functions Blocks dentro de Function Blocks 
	// Resultados da POUs CheckProfibusIOs:
	dwSlave5DigIOsErrors:				DWORD; // NX5001_1 e 2 - PO5065 addr 5
	dwSlave5Unavailable:				DWORD;
	dwSlave5ModulesOut:					DWORD;
	dwSlave10AnaIOsErrors:				DWORD; // NX5001_1 e 2 - PO5065 addr 10
	dwSlave10Unavailable:				DWORD;
	dwSlave10ModulesOut:				DWORD;
	dwSlave3DigIOsErrors:				DWORD; // NX5001_3 - PO5063 addr 4
	dwSlave3Unavailable:				DWORD;	
	dwSlave3ModulesOut:					DWORD;
	wErrorValuePO1212C00:				WORD;
	wErrorValuePO2132C00:				WORD;
	bFrozenErrorRem05TORem05:			BOOL;
	bFrozenErrorRem05TORem04:			BOOL;
	
	
	// Resultados da POU CheckModbus1:
	bModbus1ErrorCoil:					BOOL;
	bModbus1ErrorStatus:				BOOL;
	bModbus1ErrorHolding:				BOOL;
	bModbus1ErrorInputReg:				BOOL;
	// Resultados da POU CheckModbus2:
	bModbus2ErrorCoil:					BOOL;
	bModbus2ErrorStatus:				BOOL;
	bModbus2ErrorHolding:				BOOL;
	bModbus2ErrorInputReg:				BOOL;
	// Resultados da POU CheckModbus3:
	bModbus3ErrorCoil:					BOOL;
	bModbus3ErrorStatus:				BOOL;
	bModbus3ErrorHolding:				BOOL;
	bModbus3ErrorInputReg:				BOOL;
	// Resultados da POU CheckModbus4:
	bModbus4ErrorCoil:					BOOL;
	bModbus4ErrorStatus:				BOOL;
	bModbus4ErrorHolding:				BOOL;
	bModbus4ErrorInputReg:				BOOL;
	// Resultados da POU CFC (testa as linguagens de programação):
	dwErrorLanguages:					DWORD;	
	// Resultados POU CheckRecipe
	dwRecipeErrors: 					DWORD;
	dwRecipeReturnError: 				DWORD;	
	// Resultados POU CheckForcing
	bForcingDiagUnset:					BOOL;
	bBoolVarNotForced:					BOOL;
	bWordVarNotForced:					BOOL;
	// Resultados da POU CheckNVL
	{attribute 'symbol' := 'read'}
	bFailNVLCommunicationJIGA01:		BOOL;			// Houve falha na comunicação NVL com esta jiga
	{attribute 'symbol' := 'read'}
	bFailNVLCommunicationJIGA02:		BOOL;			// Houve falha na comunicação NVL com esta jiga
	{attribute 'symbol' := 'read'}
	bFailNVLCommunicationJIGA05:		BOOL;			// Houve falha na comunicação NVL com esta jiga
	{attribute 'symbol' := 'read'}
	bFailNVLCommunicationJIGA07:		BOOL;			// Houve falha na comunicação NVL com esta jiga
	
	// Eventos SOE - Não faz parte do relatório dos testes. Não modificar.
	IEC_SOE_QUEUE_INFO: SOE_QUEUE_INFO_T;

END_VAR

// Device/Application/UserGVLs/Non-Redundant/ATs
{attribute 'qualified_only'}
VAR_GLOBAL
	// 48kB de dados redundantes %Q
	aiRedundantArrayQ AT %QW16384 : ARRAY [1..12228] OF INT;
	aiRedundantArrayQ1 AT %QW28612 : ARRAY [1..12228] OF INT;
	// 48kB de dados redundantes %M
	aiRedundantArrayM AT %MW0 : ARRAY [1..12228] OF INT;
	aiRedundantArrayM1 AT %MW12228 : ARRAY [1..12228] OF INT;
	// 48kB de dados redundantes %I
	aiRedundantArrayI AT %IW16384 : ARRAY [1..12228] OF INT;
	aiRedundantArrayI1 AT %IW28612 : ARRAY [1..12228] OF INT;
	// Leitura de coils
	abyModbus1CoilsRead AT %IB68000 : ARRAY [0..119] OF BYTE;
	// Leitura de input status
	abyModbus1StatusRead AT %IB68240 : ARRAY [0..119] OF BYTE;
	// Leitura de holding registers
	awModbus1HoldingRead AT %IW68480 : ARRAY [0..119] OF WORD;
	// Leitura de input register
	awModbus1InputRegRead AT %IW68720 : ARRAY [0..119] OF WORD;
	// Escrita de coils
	abyModbus1CoilsWrite AT %QB68000 : ARRAY [0..119] OF BYTE;
	// Escrita de holding registers
	awModbus1HoldingWrite AT %QB68240 : ARRAY [0..119] OF WORD;
	abyModbus1Coils AT %QB68480 : ARRAY [0..119] OF BYTE;
	abyModbus1Status AT %QB68720 : ARRAY [0..119] OF BYTE;
	awModbus1Holding AT %QB68960 : ARRAY [0..119] OF WORD;
	awModbus1InputReg AT %QB69200 : ARRAY [0..119] OF WORD;
	// Leitura de coils
	abyModbus2CoilsRead AT %IB3320 : ARRAY [0..119] OF BYTE;
	// Leitura de holding registers
	awModbus2HoldingRead AT %IW1000 : ARRAY [0..119] OF WORD;
	// Leitura de input status
	abyModbus2StatusRead AT %IB3800 : ARRAY [0..119] OF BYTE;
	// Leitura de input register
	awModbus2InputRegRead AT %IW3560 : ARRAY [0..119] OF WORD;
	// Escrita de coils
	abyModbus2CoilsWrite AT %QB7260 : ARRAY [0..119] OF BYTE;
	// Escrita de holding registers
	awModbus2HoldingWrite AT %QW7020 : ARRAY [0..119] OF WORD;

	abyModbus2Coils AT %QB7740 : ARRAY [0..239] OF BYTE;
	abyModbus2Status AT %QB8220 : ARRAY [0..239] OF BYTE;
	awModbus2Holding AT %QB7500 : ARRAY [0..119] OF WORD;
	awModbus2InputReg AT %QB7980 : ARRAY [0..119] OF WORD;
	// Leitura de coils
	abyModbus3CoilsRead AT %IB2600 : ARRAY [0..119] OF BYTE;
	// Leitura de holding registers
	awModbus3HoldingRead AT %IW2360 : ARRAY [0..119] OF WORD;
	// Leitura de input status
	abyModbus3StatusRead AT %IB3080 : ARRAY [0..119] OF BYTE;
	// Leitura de input register
	awModbus3InputRegRead AT %IW2840 : ARRAY [0..119] OF WORD;
	// Escrita de coils
	abyModbus3CoilsWrite AT %QB6292 : ARRAY [0..119] OF BYTE;
	// Escrita de holding registers
	awModbus3HoldingWrite AT %QW6052 : ARRAY [0..119] OF WORD;
	abyModbus3Coils AT %QB5332 : ARRAY [0..239] OF BYTE;
	abyModbus3Status AT %QB5812 : ARRAY [0..239] OF BYTE;
	awModbus3Holding AT %QB5092 : ARRAY [0..119] OF WORD;
	awModbus3InputReg AT %QB5572 : ARRAY [0..119] OF WORD;
	// Utilizadas na POU CheckSoe
	bSOEPoint000 AT %QX0.0 : BOOL;
	bSOEPoint999 AT %QX999.7 : BOOL;
END_VAR

// Device/Application/UserGVLs/Non-Redundant/ProjectConstants
VAR_GLOBAL CONSTANT
	// Intervalo configurado para a tarefa MainTask [ms]
	iMainTaskInterval : INT := 250;
	// RTU COM2/COM1
	iModbus1ReadWriteDelay : INT := 9000;
	// TCP NX5000/NET1 
	iModbus2ReadWriteDelay : INT := 3250;
	// TCP NX5000/NX5000		/// JDM: 3000 deveria ser suficiente!
	iModbus3ReadWriteDelay : INT := 6000;
	// TCP NET/NX5000			/// NLT: 3000 deveria ser suficiente!
	iModbus4ReadWriteDelay : INT := 12000;
	// Tempo entre alterar o valor Profibus a ser escrito e checar o lido [ms]
	// Deve considerar o intervalo da MainTask e o atraso/filtro dos módulos.
	iProfibusDelayDigital : INT := iMainTaskInterval;
	iProfibusDelayAnalog : INT := (iMainTaskInterval + 20);
	iProfibusDelayNX : INT := (iMainTaskInterval + 20);
	// Tempo entre testes de sincronismo SNTP [ms]
	liClockSyncDelay : LINT := ((60 * 60) * 1000);
	// Tamanho da fila de eventos do servidor SOE
	wSoeEventQueueSize : WORD := 1000;
	// Informa de quanto em quanto milisegundos a taxa de comunicação MODBUS deve ser calculada
	iMsToComputeComRate : INT := 3000;
	// Divisor da quantidade total de dados redundantes a serem checados por ciclo (CheckRedData).
	// Dividir por um dos seguintes valores: 1, 2, 4, 8, 16, 32, 64, 128, 256, 512 ou 1024 (máximo).
	// O valor 1 significa consistir todos os dados em um ciclo. O valor 2 significa consistir
	// metade dos dados por ciclo. O valor 4 significa consisitir 1/4 dos dados por ciclo. Etc.
	dwCheckRedDataDivisor : DWORD := 4;
	// Valor limite de incremento das variáveis redundantes
	iValueRedLimit : INT := 20000;
	// Tempo a desconsiderar os diagnósticos quando o PLC assumir como ativo, permitindo o
	// estabelecimento e estabilização da comunicação MODBUS/Profibus [ms]
	iTimeToSkipAsActive : INT := 5000;
	// Tempo de emitir aviso antes de ocorrer o switch-over [ms] (Symbolics.byStateChangeState = 2)
	iTimeToWarnBeforeSwitchOver : INT := 2000;
	// Total: depende do modelo de UCP
	dwRamTotal : DWORD := 130289664;
	// Diferença máxima aceita entre mín/máx
	dwRamVariance : DWORD := (2 * 1024);
	// Limite para contadores do tipo INT 
	iFailCounterLimit : INT := 32767;
	// Valor enviado via NVL para informar que houve um comando de CleanTest nesta jiga
	iNVL_CleanTest : INT := -1;
	// Intervalo de tempo usado no NVL para acusar erro de comunicação [ms]
	iNVL_MaximumInterval : INT := 5000;
	// Profibus State Change, Valores limites para troca de estado
	iLowLimit : INT := 9000;
	iHighLimit : INT := 25000;
END_VAR

// Device/Application/UserGVLs/Non-Redundant/ModbusSymbol
{attribute 'qualified_only'}
VAR_GLOBAL
	// Leitura de coils
	abModbus4CoilsRead : ARRAY [0..1919] OF BOOL;
	// Leitura de holding registers
	awModbus4HoldingRead : ARRAY [0..119] OF WORD;
	// Leitura de input status
	abModbus4StatusRead : ARRAY [0..1919] OF BOOL;
	// Leitura de input registers
	awModbus4InputRegRead : ARRAY [0..119] OF WORD;
	// Escrita de coils
	abModbus4CoilsWrite : ARRAY [0..1919] OF BOOL;
	// Escrita de holding registers
	awModbus4HoldingWrite : ARRAY [0..119] OF WORD;
	abModbus4Coils : ARRAY [0..1919] OF BOOL;
	abModbus4Status : ARRAY [0..1919] OF BOOL;
	awModbus4Holding : ARRAY [0..119] OF WORD;
	awModbus4InputReg : ARRAY [0..119] OF WORD;
END_VAR

// Device/Application/UserGVLs/Non-Redundant/NonRedData
{attribute 'qualified_only'}
VAR_GLOBAL
	// Utilizado no UserLog
	iStepUserlog : INT := 0;
	// Utilizado no UserLog
	tMinimumTime : TIME := TIME#2880m0s0ms;
	// Últimos estados de redundância do PLC, ciclo a ciclo (índice 0 = ciclo atual)
	aeLastRedState : ARRAY [0..2] OF REDUNDANCY_STATE := [3(REDUNDANCY_STATE.NOT_CONFIGURED)];
	bSoeFirstCheckCycle : BOOL;
	// Temporizador para consistência dos valores Profibus
	iProfibus5DigTimer : INT := 0;
	iProfibus10AnaTimer : INT := 0;
	iProfibus3DigTimer : INT := 0;
	iProfibusNXTimer : INT := 0;
	iProfibus99AnaTimer : INT := 0;
	iProfibus99DigTimer : INT := 0;
	iProfibus99Dig1005Timer : INT := 0;
	iProfibus98DigTimer : INT := 0;
	// Indicador de mudança de estado da redundância
	bRedStateChanged : BOOL;
	{attribute 'symbol' := 'read'}
	// Indica se está no horário de verão (TRUE) ou não (FALSE)
	bDaylightSavingTime:		BOOL;
	// Horário da UCP no momento da chamada da NonSkippedPrg
	xNonSkippedPrgDateAndTime:	NextoStandard.EXTENDED_DATE_AND_TIME;
END_VAR

// Device/Application/UserGVLs/Non-Redundant/MinMaxTimes
{attribute 'qualified_only'}
VAR_GLOBAL
	// Tempo mínimo da NonSkippedPrg [us]
	uliPouMinTime_NonSkippedPrg : ULINT := 65535;
	// Tempo médio da NonSkippedPrg [us]
	uliPouAvgTime_NonSkippedPrg : ULINT;
	// Tempo máximo da NonSkippedPrg [us]
	uliPouMaxTime_NonSkippedPrg : ULINT := 0;
	// Tempo mínimo da ActivePrg [us]
	uliPouMinTime_ActivePrg : ULINT := 65535;
	// Tempo médio da ActivePrg [us]
	uliPouAvgTime_ActivePrg : ULINT;
	// Tempo máximo da ActivePrg [us]
	uliPouMaxTime_ActivePrg : ULINT := 0;
	// Soma dos tempos MÍNIMOS das POUs [us]
	uliPouMinTime_TOTAL : ULINT;
	// Soma dos tempos MÁXIMOS das POUs [us]
	uliPouMaxTime_TOTAL : ULINT;
	// Tempos mínimos/máximos de duração das POUs (lembrar de atualizar o TOTAL quando inserir/remover uma POU)
	uliPouMinTime_Alarms : ULINT := 65535;
	uliPouMaxTime_Alarms : ULINT := 0;
	uliPouMinTime_CheckIec104 : ULINT := 65535;
	uliPouMaxTime_CheckIec104 : ULINT := 0;
	uliPouMinTime_CheckLanguages : ULINT := 65535;
	uliPouMaxTime_CheckLanguages : ULINT := 0;
	uliPouMinTime_CheckModbus1 : ULINT := 65535;
	uliPouMaxTime_CheckModbus1 : ULINT := 0;
	uliPouMinTime_CheckModbus2 : ULINT := 65535;
	uliPouMaxTime_CheckModbus2 : ULINT := 0;
	uliPouMinTime_CheckModbus3 : ULINT := 65535;
	uliPouMaxTime_CheckModbus3 : ULINT := 0;
	uliPouMinTime_CheckModbus4 : ULINT := 65535;
	uliPouMaxTime_CheckModbus4 : ULINT := 0;
	uliPouMinTime_CheckProfibusIOs : ULINT := 65535;
	uliPouMaxTime_CheckProfibusIOs : ULINT := 0;
	uliPouMinTime_CheckRecipe : ULINT := 65535;
	uliPouMaxTime_CheckRecipe : ULINT := 0;
	uliPouMinTime_CheckRedData : ULINT := 65535;
	uliPouMaxTime_CheckRedData : ULINT := 0;
	uliPouMinTime_CheckSntp : ULINT := 65535;
	uliPouMaxTime_CheckSntp : ULINT := 0;
	uliPouMinTime_CheckSoe : ULINT := 65535;
	uliPouMaxTime_CheckSoe : ULINT := 0;
	uliPouMinTime_CheckSpecialVars : ULINT := 65535;
	uliPouMaxTime_CheckSpecialVars : ULINT := 0;
	uliPouMinTime_CleanStatus : ULINT := 65535;
	uliPouMaxTime_CleanStatus : ULINT := 0;
	uliPouMinTime_CycleTimes : ULINT := 65535;
	uliPouMaxTime_CycleTimes : ULINT := 0;
	uliPouMinTime_CheckDiags : ULINT := 65535;
	uliPouMaxTime_CheckDiags : ULINT := 0;
	uliPouMinTime_DaylightSavingTime : ULINT := 65535;
	uliPouMaxTime_DaylightSavingTime : ULINT := 0;
	uliPouMinTime_IncrRedData : ULINT := 65535;
	uliPouMaxTime_IncrRedData : ULINT := 0;
	uliPouMinTime_PidGenerator : ULINT := 65535;
	uliPouMaxTime_PidGenerator : ULINT := 0;
	uliPouMinTime_ProfibusStateChange : ULINT := 65535;
	uliPouMaxTime_ProfibusStateChange : ULINT := 0;
	uliPouMinTime_StateChange : ULINT := 65535;
	uliPouMaxTime_StateChange : ULINT := 0;
	uliPouMinTime_UserLog : ULINT := 65535;
	uliPouMaxTime_UserLog : ULINT := 0;
	uliPouMinTime_CheckRam : ULINT := 65535;
	uliPouMaxTime_CheckRam : ULINT := 0;
	uliPouMinTime_CheckForcing : ULINT := 65535;
	uliPouMaxTime_CheckForcing : ULINT := 0;
	uliPouMinTime_WriteHwVersionsNonActive : ULINT := 65535;
	uliPouMaxTime_WriteHwVersionsNonActive : ULINT := 0;
	uliPouMinTime_CheckNVL : ULINT := 65535;
	uliPouMaxTime_CheckNVL : ULINT := 0;
	uliPouMinTime_MQTT : ULINT := 65535;
	uliPouMaxTime_MQTT : ULINT := 0;
	// Tempos MÁXIMOS de transição das entradas que são imagem/cópia das saídas
	liDigMaxTime_CheckModbus1 : LINT := 0;
	liAnaMaxTime_CheckModbus1 : LINT := 0;
	liDigMaxTime_CheckModbus2 : LINT := 0;
	liAnaMaxTime_CheckModbus2 : LINT := 0;
	liDigMaxTime_CheckModbus3 : LINT := 0;
	liAnaMaxTime_CheckModbus3 : LINT := 0;
	liDigMaxTime_CheckModbus4 : LINT := 0;
	liAnaMaxTime_CheckModbus4 : LINT := 0;
	liDigMaxTime_CheckProfibusIOs : LINT := 0;
	liAnaMaxTime_CheckProfibusIOs : LINT := 0;
	liNXMaxTime_CheckProfibusIOs : LINT := 0;
	liAna99MaxTime_CheckProfibusIOs : LINT := 0;
	liDig99MaxTime_CheckProfibusIOs : LINT := 0;
	liDig99MaxTime1005_CheckProfibusIOs : LINT := 0;
	// Taxas médias de comunicação MODBUS [Bytes/Second]
	diModbus1BytesPerSec : DINT;
	diModbus2BytesPerSec : DINT;
	diModbus3BytesPerSec : DINT;
	diModbus4BytesPerSec : DINT;
	// Variáveis para depuração do BUG 19183
	{attribute '''DOCU__COMMENT' := ' Variáveis para depuração do BUG 19183'}
	auliRedRemainTimeoutCounter : ARRAY [0..99] OF ULINT;
END_VAR

// Device/Application/UserGVLs/Non-Redundant/DiagsRetain
{attribute 'qualified_only'}
VAR_GLOBAL RETAIN
	// NX3030
	DG_NX3030_tSummarized_bAbsentModules : BOOL;
	DG_NX3030_tSummarized_bAbsentRacks : BOOL;
	DG_NX3030_tSummarized_bCOM1ConfigError : BOOL;
	DG_NX3030_tSummarized_bCOM2ConfigError : BOOL;
	DG_NX3030_tSummarized_bConfigMismatch : BOOL;
	DG_NX3030_tSummarized_bDuplicatedRacks : BOOL;
	DG_NX3030_tSummarized_bDuplicatedSlots : BOOL;
	DG_NX3030_tSummarized_bHardwareFailure : BOOL;
	DG_NX3030_tSummarized_bInvalidDateTime : BOOL;
	DG_NX3030_tSummarized_bInvalidRacks : BOOL;
	DG_NX3030_tSummarized_bMemoryCardError : BOOL;
	DG_NX3030_tSummarized_bModuleFatalError : BOOL;
	DG_NX3030_tSummarized_bModuleParameterError : BOOL;
	DG_NX3030_tSummarized_bModulesWithDiagnostic : BOOL;
	DG_NX3030_tSummarized_bNET1ConfigError : BOOL;
	DG_NX3030_tSummarized_bNET2ConfigError : BOOL;
	DG_NX3030_tSummarized_bNonDeclaredModules : BOOL;
	DG_NX3030_tSummarized_bNonDeclaredRacks : BOOL;
	DG_NX3030_tSummarized_bOTDSwitchError : BOOL;
	DG_NX3030_tSummarized_bRuntimeReset : BOOL;
	DG_NX3030_tSummarized_bSoftwareException : BOOL;
	DG_NX3030_tSummarized_bSwappedModules : BOOL;
	DG_NX3030_tSummarized_bWHSBBusError : BOOL;
	DG_NX3030_tDetailed_MemoryCard_byMounted : BOOL;
	DG_NX3030_tDetailed_Ethernet_NET1_bLinkDown : BOOL;
	DG_NX3030_tDetailed_Ethernet_NET2_bLinkDown : BOOL;
	DG_NX3030_tDetailed_Application_byCPUState : BOOL;
	DG_NX3030_tDetailed_ApplicationInfo_dwApplicationCRC : BOOL;
	DG_NX3030_tDetailed_Ethernet_NET1_abyMAC_0 : BOOL;
	DG_NX3030_tDetailed_Ethernet_NET1_abyMAC_1 : BOOL;
	DG_NX3030_tDetailed_Ethernet_NET1_abyMAC_2 : BOOL;
	DG_NX3030_tDetailed_Ethernet_NET1_abyMAC_3 : BOOL;
	DG_NX3030_tDetailed_Ethernet_NET1_abyMAC_4 : BOOL;
	DG_NX3030_tDetailed_Ethernet_NET1_abyMAC_5 : BOOL;
	DG_NX3030_tDetailed_Ethernet_NET2_abyMAC_0 : BOOL;
	DG_NX3030_tDetailed_Ethernet_NET2_abyMAC_1 : BOOL;
	DG_NX3030_tDetailed_Ethernet_NET2_abyMAC_2 : BOOL;
	DG_NX3030_tDetailed_Ethernet_NET2_abyMAC_3 : BOOL;
	DG_NX3030_tDetailed_Ethernet_NET2_abyMAC_4 : BOOL;
	DG_NX3030_tDetailed_Ethernet_NET2_abyMAC_5 : BOOL;
	DG_NX3030_tDetailed_Ethernet_NETx_abyIP_0 : BOOL;
	DG_NX3030_tDetailed_Ethernet_NETx_abyIP_1 : bool;
	DG_NX3030_tDetailed_Ethernet_NETx_abyIP_2 : bool;
	DG_NX3030_tDetailed_Ethernet_NETx_abyIP_3 : bool;
	DG_NX3030_tDetailed_Ethernet_NETx_abyMask_0 : bool;
	DG_NX3030_tDetailed_Ethernet_NETx_abyMask_1 : bool;
	DG_NX3030_tDetailed_Ethernet_NETx_abyMask_2 : bool;
	DG_NX3030_tDetailed_Ethernet_NETx_abyMask_3 : bool;
	DG_NX3030_tDetailed_Ethernet_NETx_abyGateway_0 : bool;
	DG_NX3030_tDetailed_Ethernet_NETx_abyGateway_1 : bool;
	DG_NX3030_tDetailed_Ethernet_NETx_abyGateway_2 : bool;
	DG_NX3030_tDetailed_Ethernet_NETx_abyGateway_3 : bool;
	DG_NX3030_tDetailed_SNTP_bServiceEnabled : bool;
	DG_NX3030_tDetailed_Target_abyAuxprocVersion : BOOL;
	DG_NX3030_tDetailed_Target_abyBootloaderVersion : BOOL;
	DG_NX3030_tDetailed_Target_abyCPUVersion : BOOL;
	DG_NX3030_tDetailed_Target_dwCPUModel : BOOL;
	DG_NX3030_tDetailed_Thermometer_diTemperature : bool;
	// NX4010
	DG_NX4010_tGeneral_bActiveDiagnostics : BOOL;
	DG_NX4010_tGeneral_bBusCommunicationError : BOOL;
	DG_NX4010_tGeneral_bConfigMismatch : BOOL;
	DG_NX4010_tGeneral_bFatalError : BOOL;
	DG_NX4010_tGeneral_bNET1LinkDown : BOOL;
	DG_NX4010_tGeneral_bNET2LinkDown : BOOL;
	DG_NX4010_tGeneral_bOTDSwitchError : BOOL;
	DG_NX4010_tGeneral_bWatchdogError : BOOL;
	DG_NX4010_tRedundancy_RedDgnLoc_sGeneral_Diag_bApplicationIncompatible : BOOL;
	DG_NX4010_tRedundancy_RedDgnLoc_sGeneral_Diag_bApplicationProjectDiff : BOOL;
	DG_NX4010_tRedundancy_RedDgnLoc_sGeneral_Diag_bConfigError : BOOL;
	DG_NX4010_tRedundancy_RedDgnLoc_sGeneral_Diag_bExchangeSync : BOOL;
	DG_NX4010_tRedundancy_RedDgnLoc_sGeneral_Diag_bFailedPBUS1A : BOOL;
	DG_NX4010_tRedundancy_RedDgnLoc_sGeneral_Diag_bFailedPBUS1B : BOOL;
	DG_NX4010_tRedundancy_RedDgnLoc_sGeneral_Diag_bFailedPBUS2A : BOOL;
	DG_NX4010_tRedundancy_RedDgnLoc_sGeneral_Diag_bFailedPBUS2B : BOOL;
	DG_NX4010_tRedundancy_RedDgnLoc_sGeneral_Diag_bFailedRED : BOOL;
	DG_NX4010_tRedundancy_RedDgnLoc_sGeneral_Diag_bFailureProfibus_1 : BOOL;
	DG_NX4010_tRedundancy_RedDgnLoc_sGeneral_Diag_bFailureProfibus_2 : BOOL;
	DG_NX4010_tRedundancy_RedDgnLoc_sGeneral_Diag_bIncompatibleFirmware : BOOL;
	DG_NX4010_tRedundancy_RedDgnLoc_sGeneral_Diag_bProfibusVitalFailureAll : BOOL;
	DG_NX4010_tRedundancy_RedDgnLoc_sGeneral_Diag_bProfibusVitalFailureAny : BOOL;
	DG_NX4010_tRedundancy_RedDgnLoc_sGeneral_Diag_bProjectArchiveDiff : BOOL;
	DG_NX4010_tRedundancy_RedDgnLoc_sGeneral_Diag_bProjectSyncDisable : BOOL;
	DG_NX4010_tRedundancy_RedDgnLoc_sGeneral_Diag_bRedDataSync : BOOL;
	DG_NX4010_tRedundancy_RedDgnLoc_sGeneral_Diag_bRedForceSync : BOOL;
	DG_NX4010_tRedundancy_RedDgnLoc_sGeneral_Diag_bRedPanelTestMode : BOOL;
	DG_NX4010_tRedundancy_RedDgnLoc_sGeneral_Diag_bTemporaryBufferTooSmall : BOOL;
	DG_NX4010_tRedundancy_RedDgnLoc_sGeneral_Diag_bTooManyRedAreas : BOOL;
	DG_NX4010_tRedundancy_RedDgnLoc_sGeneral_Diag_dwApplicationCRC : BOOL;
	DG_NX4010_tRedundancy_RedDgnLoc_sGeneral_Diag_dwArchiveCRC : BOOL;
	// NX5001_1
	DG_NX5001_1_tGeneral_bActiveDiagnostics : BOOL;
	DG_NX5001_1_tGeneral_bBusCommunicationError : BOOL;
	DG_NX5001_1_tGeneral_bConfigMismatch : BOOL;
	DG_NX5001_1_tGeneral_bFatalError : BOOL;
	DG_NX5001_1_tGeneral_bNX5001NoCfg : BOOL;
	DG_NX5001_1_tGeneral_bOTDSwitchError : BOOL;
	DG_NX5001_1_tGeneral_bPbusCommFail : BOOL;
	DG_NX5001_1_tGeneral_bSlaveNotConfigured : BOOL;
	DG_NX5001_1_tGeneral_bSlaveNotPresent : BOOL;
	DG_NX5001_1_tGeneral_bSlaveWithDiagnostic : BOOL;
	DG_NX5001_1_tGeneral_bStsEnableInterface : BOOL;
	DG_NX5001_1_tGeneral_bStsMstRedundEnable : BOOL;
	DG_NX5001_1_tGeneral_bWatchdogError : BOOL;
	DG_NX5001_1_tMstStatus_abySlv_Diag_bSlave_5 : BOOL;
	DG_NX5001_1_tMstStatus_abySlv_Diag_bSlave_10 : BOOL;
	DG_NX5001_1_tMstStatus_abySlv_Diag_bSlave_99 : BOOL;
	// NX5001_2
	DG_NX5001_2_tGeneral_bActiveDiagnostics : BOOL;
	DG_NX5001_2_tGeneral_bBusCommunicationError : BOOL;
	DG_NX5001_2_tGeneral_bConfigMismatch : BOOL;
	DG_NX5001_2_tGeneral_bFatalError : BOOL;
	DG_NX5001_2_tGeneral_bNX5001NoCfg : BOOL;
	DG_NX5001_2_tGeneral_bOTDSwitchError : BOOL;
	DG_NX5001_2_tGeneral_bPbusCommFail : BOOL;
	DG_NX5001_2_tGeneral_bSlaveNotConfigured : BOOL;
	DG_NX5001_2_tGeneral_bSlaveNotPresent : BOOL;
	DG_NX5001_2_tGeneral_bSlaveWithDiagnostic : BOOL;
	DG_NX5001_2_tGeneral_bStsEnableInterface : BOOL;
	DG_NX5001_2_tGeneral_bStsMstRedundEnable : BOOL;
	DG_NX5001_2_tGeneral_bWatchdogError : BOOL;
	DG_NX5001_2_tMstStatus_abySlv_Diag_bSlave_5 : BOOL;
	DG_NX5001_2_tMstStatus_abySlv_Diag_bSlave_10 : BOOL;
	DG_NX5001_2_tMstStatus_abySlv_Diag_bSlave_99 : BOOL;
	// NX5001_3
	DG_NX5001_3_tGeneral_bActiveDiagnostics : BOOL;
	DG_NX5001_3_tGeneral_bBusCommunicationError : BOOL;
	DG_NX5001_3_tGeneral_bConfigMismatch : BOOL;
	DG_NX5001_3_tGeneral_bFatalError : BOOL;
	DG_NX5001_3_tGeneral_bNX5001NoCfg : BOOL;
	DG_NX5001_3_tGeneral_bOTDSwitchError : BOOL;
	DG_NX5001_3_tGeneral_bPbusCommFail : BOOL;
	DG_NX5001_3_tGeneral_bSlaveNotConfigured : BOOL;
	DG_NX5001_3_tGeneral_bSlaveNotPresent : BOOL;
	DG_NX5001_3_tGeneral_bSlaveWithDiagnostic : BOOL;
	DG_NX5001_3_tGeneral_bStsEnableInterface : BOOL;
	DG_NX5001_3_tGeneral_bStsMstRedundEnable : BOOL;
	DG_NX5001_3_tGeneral_bWatchdogError : BOOL;
	DG_NX5001_3_tMstStatus_abySlv_Diag_bSlave_4 : BOOL;
	DG_NX5001_3_tMstStatus_abySlv_Diag_bSlave_99 : BOOL;
	// NX5000_1	
	DG_NX5000_1_tGeneral_bActiveDiagnostics : BOOL;
	DG_NX5000_1_tGeneral_bBusCommunicationError : BOOL;
	DG_NX5000_1_tGeneral_bConfigMismatch : BOOL;
	DG_NX5000_1_tGeneral_bFatalError : BOOL;
	DG_NX5000_1_tGeneral_bOTDSwitchError : BOOL;
	DG_NX5000_1_tGeneral_bWatchdogError : BOOL;
	DG_NX5000_1_tNX5000_bNX5000NoCfg : BOOL;
	DG_NX5000_1_tNX5000_bStsEthLink : BOOL;
	// NX5000_2	
	DG_NX5000_2_tGeneral_bActiveDiagnostics : BOOL;
	DG_NX5000_2_tGeneral_bBusCommunicationError : BOOL;
	DG_NX5000_2_tGeneral_bConfigMismatch : BOOL;
	DG_NX5000_2_tGeneral_bFatalError : BOOL;
	DG_NX5000_2_tGeneral_bOTDSwitchError : BOOL;
	DG_NX5000_2_tGeneral_bWatchdogError : BOOL;
	DG_NX5000_2_tNX5000_bNX5000NoCfg : BOOL;
	DG_NX5000_2_tNX5000_bStsEthLink : BOOL;
	// NX5000_3	
	DG_NX5000_3_tGeneral_bActiveDiagnostics : BOOL;
	DG_NX5000_3_tGeneral_bBusCommunicationError : BOOL;
	DG_NX5000_3_tGeneral_bConfigMismatch : BOOL;
	DG_NX5000_3_tGeneral_bFatalError : BOOL;
	DG_NX5000_3_tGeneral_bOTDSwitchError : BOOL;
	DG_NX5000_3_tGeneral_bWatchdogError : BOOL;
	DG_NX5000_3_tNX5000_bNX5000NoCfg : BOOL;
	DG_NX5000_3_tNX5000_bStsEthLink : BOOL;
	// DG_MODBUS_Master_1
	DG_MODBUS_Master_1_tDiag_bConfigFailure : BOOL;
	DG_MODBUS_Master_1_tDiag_bModuleFailure : BOOL;
	DG_MODBUS_Master_1_tDiag_bRXFailure : BOOL;
	DG_MODBUS_Master_1_tDiag_bTXFailure : BOOL;
	// MODBUS_Slave_1	
	DG_MODBUS_Slave_1_tDiag_bConfigFailure : BOOL;
	DG_MODBUS_Slave_1_tDiag_bModuleFailure : BOOL;
	DG_MODBUS_Slave_1_tDiag_bRXFailure : BOOL;
	DG_MODBUS_Slave_1_tDiag_bTXFailure : BOOL;
	// MODBUS_Client_2
	DG_MODBUS_Client_2_tDiag_bConfigFailure : BOOL;
	DG_MODBUS_Client_2_tDiag_bModuleFailure : BOOL;
	DG_MODBUS_Client_2_tDiag_bRXFailure : BOOL;
	DG_MODBUS_Client_2_tDiag_bTXFailure : BOOL;
	// MODBUS_Server_2
	DG_MODBUS_Server_2_tDiag_bConfigFailure : BOOL;
	DG_MODBUS_Server_2_tDiag_bModuleFailure : BOOL;
	DG_MODBUS_Server_2_tDiag_bRXFailure : BOOL;
	DG_MODBUS_Server_2_tDiag_bTXFailure : BOOL;
	// MODBUS_Client_3
	DG_MODBUS_Client_3_tDiag_bConfigFailure : BOOL;
	DG_MODBUS_Client_3_tDiag_bModuleFailure : BOOL;
	DG_MODBUS_Client_3_tDiag_bRXFailure : BOOL;
	DG_MODBUS_Client_3_tDiag_bTXFailure : BOOL;
	// MODBUS_Server_3
	DG_MODBUS_Server_3_tDiag_bConfigFailure : BOOL;
	DG_MODBUS_Server_3_tDiag_bModuleFailure : BOOL;
	DG_MODBUS_Server_3_tDiag_bRXFailure : BOOL;
	DG_MODBUS_Server_3_tDiag_bTXFailure : BOOL;
	// MODBUS_Client_4
	DG_MODBUS_Client_4_tDiag_bConfigFailure : BOOL;
	DG_MODBUS_Client_4_tDiag_bModuleFailure : BOOL;
	DG_MODBUS_Client_4_tDiag_bRXFailure : BOOL;
	DG_MODBUS_Client_4_tDiag_bTXFailure : BOOL;
	// MODBUS_Server_4	
	DG_MODBUS_Server_4_tDiag_bConfigFailure : BOOL;
	DG_MODBUS_Server_4_tDiag_bModuleFailure : BOOL;
	DG_MODBUS_Server_4_tDiag_bRXFailure : BOOL;
	DG_MODBUS_Server_4_tDiag_bTXFailure : BOOL;

	//PO1000
	DG_REM05_PO1000_bHardwareFailure : bool;
	DG_REM05_PO1000_bPowerSupplyFail : bool;
	
	//PO2020
	DG_REM05_PO2020_bHardwareFailure : bool;
	DG_REM05_PO2020_bPowerSupplyFail : bool;

	//PO9100	
	DG_REM05_PO9100_bReserved00 : bool;
	
	//PO1212
	DG_REM10_PO1212_bFuseOpen : bool;
	DG_REM10_PO1212_bHardwareFailure : bool;
	DG_REM10_PO1212_bNoParametrizedModule : bool;
	DG_REM10_PO1212_bOverTemp : bool;
	DG_REM10_PO1212_aCh0_bOpenSensor : bool;
	DG_REM10_PO1212_aCh0_bOverRange : bool;
	DG_REM10_PO1212_aCh0_bSensorShortCircuit : bool;
	DG_REM10_PO1212_aCh0_bWrongParameters : bool;
	DG_REM10_PO1212_aCh1_bOpenSensor : bool;
	DG_REM10_PO1212_aCh1_bOverRange : bool;
	DG_REM10_PO1212_aCh1_bSensorShortCircuit : bool;
	DG_REM10_PO1212_aCh1_bWrongParameters : bool;
	DG_REM10_PO1212_aCh2_bOpenSensor : bool;
	DG_REM10_PO1212_aCh2_bOverRange : bool;
	DG_REM10_PO1212_aCh2_bSensorShortCircuit : bool;
	DG_REM10_PO1212_aCh2_bWrongParameters : bool;
	DG_REM10_PO1212_aCh3_bOpenSensor : bool;
	DG_REM10_PO1212_aCh3_bOverRange : bool;
	DG_REM10_PO1212_aCh3_bSensorShortCircuit : bool;
	DG_REM10_PO1212_aCh3_bWrongParameters : bool;
	DG_REM10_PO1212_aCh4_bOpenSensor : bool;
	DG_REM10_PO1212_aCh4_bOverRange : bool;
	DG_REM10_PO1212_aCh4_bSensorShortCircuit : bool;
	DG_REM10_PO1212_aCh4_bWrongParameters : bool;
	DG_REM10_PO1212_aCh5_bOpenSensor : bool;
	DG_REM10_PO1212_aCh5_bOverRange : bool;
	DG_REM10_PO1212_aCh5_bSensorShortCircuit : bool;
	DG_REM10_PO1212_aCh5_bWrongParameters : bool;
	DG_REM10_PO1212_aCh6_bOpenSensor : bool;
	DG_REM10_PO1212_aCh6_bOverRange : bool;
	DG_REM10_PO1212_aCh6_bSensorShortCircuit : bool;
	DG_REM10_PO1212_aCh6_bWrongParameters : bool;
	DG_REM10_PO1212_aCh7_bOpenSensor : bool;
	DG_REM10_PO1212_aCh7_bOverRange : bool;
	DG_REM10_PO1212_aCh7_bSensorShortCircuit : bool;
	DG_REM10_PO1212_aCh7_bWrongParameters : bool;
	
	//PO2132
	DG_REM10_PO2132_bNoParametrizedModule : bool;
	DG_REM10_PO2132_bPowerSupplyFail : bool;
	DG_REM10_PO2132_aCh0_bOpenSensor : bool;
	DG_REM10_PO2132_aCh0_bWrongParameters : bool;
	DG_REM10_PO2132_aCh1_bOpenSensor : bool;
	DG_REM10_PO2132_aCh1_bWrongParameters : bool;
	DG_REM10_PO2132_aCh2_bOpenSensor : bool;
	DG_REM10_PO2132_aCh2_bWrongParameters : bool;
	DG_REM10_PO2132_aCh3_bOpenSensor : bool;
	DG_REM10_PO2132_aCh3_bWrongParameters : bool;

	
	//PO9100
	DG_REM10_PO9100_bReserved00 : bool;
	
	//PO1000
	DG_REM04_PO1000_bHardwareFailure : bool;
	DG_REM04_PO1000_bPowerSupplyFail : bool;
	
	
END_VAR

// Device/Application/UserGVLs/Non-Redundant/HwVersions
{attribute 'qualified_only'}
VAR_GLOBAL
	{attribute 'symbol' := 'read'}
	eR00S02_NX3030_PlcA : Firmware_CPU;
	{attribute 'symbol' := 'read'}
	eR00S04_NX4010_PlcA : Firmware;
	{attribute 'symbol' := 'read'}
	eR00S06_NX5001_PlcA : Firmware;
	{attribute 'symbol' := 'read'}
	eR00S08_NX5001_PlcA : Firmware;
	{attribute 'symbol' := 'read'}
	eR00S10_NX5000_PlcA : Firmware;
	{attribute 'symbol' := 'read'}
	eR00S12_NX5000_PlcA : Firmware;
	{attribute 'symbol' := 'read'}
	eR00S16_NX5001_PlcA : Firmware;
	{attribute 'symbol' := 'read'}
	eR00S20_NX5000_PlcA : Firmware;
	{attribute 'symbol' := 'read'}
	eR00S02_NX3030_PlcB : Firmware_CPU;
	{attribute 'symbol' := 'read'}
	eR00S04_NX4010_PlcB : Firmware;
	{attribute 'symbol' := 'read'}
	eR00S06_NX5001_PlcB : Firmware;
	{attribute 'symbol' := 'read'}
	eR00S08_NX5001_PlcB : Firmware;
	{attribute 'symbol' := 'read'}
	eR00S10_NX5000_PlcB : Firmware;
	{attribute 'symbol' := 'read'}
	eR00S12_NX5000_PlcB : Firmware;
	{attribute 'symbol' := 'read'}
	eR00S16_NX5001_PlcB : Firmware;
	{attribute 'symbol' := 'read'}
	eR00S20_NX5000_PlcB : Firmware;
END_VAR

// Device/Application/UserGVLs/Non-Redundant/Task_Information
{attribute 'qualified_only'}
VAR_GLOBAL RETAIN
	// Esta GVL contêm os dados de cada tarefa que o Sistema apresenta no Task Monitor
	TI_MainTask : Task_Informations;
	TI_Configuration : Task_Informations;
	TI_MODBUS_Client_2 : Task_Informations;
	TI_MODBUS_Client_3 : Task_Informations;
	TI_MODBUS_Master_1 : Task_Informations;
	TI_MODBUS_Server_2 : Task_Informations;
	TI_MODBUS_Server_3 : Task_Informations;
	TI_MODBUS_Slave_1 : Task_Informations;
END_VAR

// Device/Application/UserGVLs/Non-Redundant/SymbolicsNonRedundant
{attribute 'qualified_only'}
VAR_GLOBAL
	// Indica comando de reinicialização das estatísticas
	bEnableCleanStats_CheckForcing : BOOL;
	// Indica comando de reinicialização das estatísticas
	bEnableCleanStats_CheckSntp : BOOL;
	// Indica comando de reinicialização das estatísticas	
	bEnableCleanStats_CheckRam : BOOL;
	// Indica comando de reinicialização das estatísticas
	bEnableCleanStats_CheckRedData : BOOL;
	// Indica comando de reinicialização das estatísticas
	bEnableCleanStats_NonSkippedPrg : BOOL;
	// Indica comando de reinicialização das estatísticas
	bEnableCleanStats_CheckDiagsRetain : BOOL;
	// Indica comando de leitura do hardware
	bReadHWVersions : BOOL;
END_VAR

// Device/Application/UserGVLs/Non-Redundant/NonRedPointer
{attribute 'qualified_only'}
VAR_GLOBAL
	// Esta GVL não deve ser retentiva devido a inicialização de ponteiros.
	// Movimentação das informações sobre o Firmware do PLC reserva para o ativo
	pdw02CPUModelRedUsrRem : POINTER TO DWORD := ADR(DG_NX4010.tRedundancy.RedUsrRem.abyUser[13]);
	pdw04NX4010FWRedUsrRem : POINTER TO DWORD := ADR(DG_NX4010.tRedundancy.RedUsrRem.abyUser[17]);
	pdw04NX4010HWRedUsrRem : POINTER TO DWORD := ADR(DG_NX4010.tRedundancy.RedUsrRem.abyUser[21]);
	pdw06NX5001FWRedUsrRem : POINTER TO DWORD := ADR(DG_NX4010.tRedundancy.RedUsrRem.abyUser[25]);
	pdw06NX5001HWRedUsrRem : POINTER TO DWORD := ADR(DG_NX4010.tRedundancy.RedUsrRem.abyUser[29]);
	pdw08NX5001FWRedUsrRem : POINTER TO DWORD := ADR(DG_NX4010.tRedundancy.RedUsrRem.abyUser[33]);
	pdw08NX5001HWRedUsrRem : POINTER TO DWORD := ADR(DG_NX4010.tRedundancy.RedUsrRem.abyUser[37]);
	pdw10NX5000FWRedUsrRem : POINTER TO DWORD := ADR(DG_NX4010.tRedundancy.RedUsrRem.abyUser[41]);
	pdw10NX5000HWRedUsrRem : POINTER TO DWORD := ADR(DG_NX4010.tRedundancy.RedUsrRem.abyUser[45]);
	pdw12NX5000FWRedUsrRem : POINTER TO DWORD := ADR(DG_NX4010.tRedundancy.RedUsrRem.abyUser[49]);
	pdw12NX5000HWRedUsrRem : POINTER TO DWORD := ADR(DG_NX4010.tRedundancy.RedUsrRem.abyUser[53]);
	pdw16NX5001FWRedUsrRem : POINTER TO DWORD := ADR(DG_NX4010.tRedundancy.RedUsrRem.abyUser[57]);
	pdw16NX5001HWRedUsrRem : POINTER TO DWORD := ADR(DG_NX4010.tRedundancy.RedUsrRem.abyUser[61]);
	pdw20NX5000FWRedUsrRem : POINTER TO DWORD := ADR(DG_NX4010.tRedundancy.RedUsrRem.abyUser[65]);
	pdw20NX5000HWRedUsrRem : POINTER TO DWORD := ADR(DG_NX4010.tRedundancy.RedUsrRem.abyUser[69]);
	pdw02CPUModelRedUsrLoc : POINTER TO DWORD := ADR(DG_NX4010.tRedundancy.RedUsrLoc.abyUser[13]);
	pdw04NX4010FWRedUsrLoc : POINTER TO DWORD := ADR(DG_NX4010.tRedundancy.RedUsrLoc.abyUser[17]);
	pdw04NX4010HWRedUsrLoc : POINTER TO DWORD := ADR(DG_NX4010.tRedundancy.RedUsrLoc.abyUser[21]);
	pdw06NX5001FWRedUsrLoc : POINTER TO DWORD := ADR(DG_NX4010.tRedundancy.RedUsrLoc.abyUser[25]);
	pdw06NX5001HWRedUsrLoc : POINTER TO DWORD := ADR(DG_NX4010.tRedundancy.RedUsrLoc.abyUser[29]);
	pdw08NX5001FWRedUsrLoc : POINTER TO DWORD := ADR(DG_NX4010.tRedundancy.RedUsrLoc.abyUser[33]);
	pdw08NX5001HWRedUsrLoc : POINTER TO DWORD := ADR(DG_NX4010.tRedundancy.RedUsrLoc.abyUser[37]);
	pdw10NX5000FWRedUsrLoc : POINTER TO DWORD := ADR(DG_NX4010.tRedundancy.RedUsrLoc.abyUser[41]);
	pdw10NX5000HWRedUsrLoc : POINTER TO DWORD := ADR(DG_NX4010.tRedundancy.RedUsrLoc.abyUser[45]);
	pdw12NX5000FWRedUsrLoc : POINTER TO DWORD := ADR(DG_NX4010.tRedundancy.RedUsrLoc.abyUser[49]);
	pdw12NX5000HWRedUsrLoc : POINTER TO DWORD := ADR(DG_NX4010.tRedundancy.RedUsrLoc.abyUser[53]);
	pdw16NX5001FWRedUsrLoc : POINTER TO DWORD := ADR(DG_NX4010.tRedundancy.RedUsrLoc.abyUser[57]);
	pdw16NX5001HWRedUsrLoc : POINTER TO DWORD := ADR(DG_NX4010.tRedundancy.RedUsrLoc.abyUser[61]);
	pdw20NX5000FWRedUsrLoc : POINTER TO DWORD := ADR(DG_NX4010.tRedundancy.RedUsrLoc.abyUser[65]);
	pdw20NX5000HWRedUsrLoc : POINTER TO DWORD := ADR(DG_NX4010.tRedundancy.RedUsrLoc.abyUser[69]);
	// Variáveis para a verificação de falha na Sincronização de Dados para ambos os Clusterss
	piSSyncFailLoc : POINTER TO INT := ADR(DG_NX4010.tRedundancy.RedUsrLoc.abyUser[73]);
	piQSyncFailLoc : POINTER TO INT := ADR(DG_NX4010.tRedundancy.RedUsrLoc.abyUser[75]);
	piMSyncFailLoc : POINTER TO INT := ADR(DG_NX4010.tRedundancy.RedUsrLoc.abyUser[77]);
	piISyncFailLoc : POINTER TO INT := ADR(DG_NX4010.tRedundancy.RedUsrLoc.abyUser[79]);
	piSSyncFailRem : POINTER TO INT := ADR(DG_NX4010.tRedundancy.RedUsrRem.abyUser[73]);
	piQSyncFailRem : POINTER TO INT := ADR(DG_NX4010.tRedundancy.RedUsrRem.abyUser[75]);
	piMSyncFailRem : POINTER TO INT := ADR(DG_NX4010.tRedundancy.RedUsrRem.abyUser[77]);
	piISyncFailRem : POINTER TO INT := ADR(DG_NX4010.tRedundancy.RedUsrRem.abyUser[79]);
	// Variáveis para a verificação de falha no SNTP para ambos os Clusters
	pbSntpServerFailuresLoc : POINTER TO BOOL := ADR(DG_NX4010.tRedundancy.RedUsrLoc.abyUser[81]);
	pbSntpSourceFailuresLoc : POINTER TO BOOL := ADR(DG_NX4010.tRedundancy.RedUsrLoc.abyUser[82]);
	piSntpSyncFailuresLoc : POINTER TO INT := ADR(DG_NX4010.tRedundancy.RedUsrLoc.abyUser[83]);
	pbSntpServerFailuresRem : POINTER TO BOOL := ADR(DG_NX4010.tRedundancy.RedUsrRem.abyUser[81]);
	pbSntpSourceFailuresRem : POINTER TO BOOL := ADR(DG_NX4010.tRedundancy.RedUsrRem.abyUser[82]);
	piSntpSyncFailuresRem : POINTER TO INT := ADR(DG_NX4010.tRedundancy.RedUsrRem.abyUser[83]);
	//  Variáveis para a verificação de falha no MODBUS Master 1 para ambos os Clusters
	pbModbus1ErrorCoilLoc : POINTER TO BOOL := ADR(DG_NX4010.tRedundancy.RedUsrLoc.abyUser[85]);
	pbModbus1ErrorStatusLoc : POINTER TO BOOL := ADR(DG_NX4010.tRedundancy.RedUsrLoc.abyUser[86]);
	pbModbus1ErrorHoldingLoc : POINTER TO BOOL := ADR(DG_NX4010.tRedundancy.RedUsrLoc.abyUser[87]);
	pbModbus1ErrorInputRegLoc : POINTER TO BOOL := ADR(DG_NX4010.tRedundancy.RedUsrLoc.abyUser[88]);
	pbModbus1ErrorCoilRem : POINTER TO BOOL := ADR(DG_NX4010.tRedundancy.RedUsrRem.abyUser[85]);
	pbModbus1ErrorStatusRem : POINTER TO BOOL := ADR(DG_NX4010.tRedundancy.RedUsrRem.abyUser[86]);
	pbModbus1ErrorHoldingRem : POINTER TO BOOL := ADR(DG_NX4010.tRedundancy.RedUsrRem.abyUser[87]);
	pbModbus1ErrorInputRegRem : POINTER TO BOOL := ADR(DG_NX4010.tRedundancy.RedUsrRem.abyUser[88]);
	//  Variáveis para a verificação de falha no Forçamento para ambos os Clusters
	// Contador de falhas no diagnóstico de forçamento
	piForcingDiagUnsetLoc : POINTER TO INT := ADR(DG_NX4010.tRedundancy.RedUsrLoc.abyUser[89]);
	piForcingDiagUnsetRem : POINTER TO INT := ADR(DG_NX4010.tRedundancy.RedUsrRem.abyUser[89]);
	// Contador de falhas de forçamento da variável BOOL
	piBoolVarNotForcedLoc : POINTER TO INT := ADR(DG_NX4010.tRedundancy.RedUsrLoc.abyUser[91]);
	piBoolVarNotForcedRem : POINTER TO INT := ADR(DG_NX4010.tRedundancy.RedUsrRem.abyUser[91]);
	// Contador de falhas de forçamento da variável WORD
	piWordVarNotForcedLoc : POINTER TO INT := ADR(DG_NX4010.tRedundancy.RedUsrLoc.abyUser[93]);
	piWordVarNotForcedRem : POINTER TO INT := ADR(DG_NX4010.tRedundancy.RedUsrRem.abyUser[93]);
	//  Variáveis para a verificação de falha no UserLog para ambos os Clusters
	pbErrorUserLogLoc : POINTER TO BOOL := ADR(DG_NX4010.tRedundancy.RedUsrLoc.abyUser[95]);
	pbErrorUserLogRem : POINTER TO BOOL := ADR(DG_NX4010.tRedundancy.RedUsrRem.abyUser[95]);
	// Indicação de falha na consistência de memória RAM total
	pbRamTotalFailureLoc : POINTER TO BOOL := ADR(DG_NX4010.tRedundancy.RedUsrLoc.abyUser[97]);
	pbRamTotalFailureRem : POINTER TO BOOL := ADR(DG_NX4010.tRedundancy.RedUsrRem.abyUser[97]);
	// Indicação de falha na consistência de memória RAM livre
	pbRamFreeVarFailureLoc : POINTER TO BOOL := ADR(DG_NX4010.tRedundancy.RedUsrLoc.abyUser[98]);
	pbRamFreeVarFailureRem : POINTER TO BOOL := ADR(DG_NX4010.tRedundancy.RedUsrRem.abyUser[98]);
	// Indicação de falha na consistência das variáveis especiais
	pbSpecialVariablesLoc : POINTER TO BOOL := ADR(DG_NX4010.tRedundancy.RedUsrLoc.abyUser[99]);
	pbSpecialVariablesRem : POINTER TO BOOL := ADR(DG_NX4010.tRedundancy.RedUsrRem.abyUser[99]);
END_VAR

// Device/Application/UserGVLs/Redundant/Languages
{attribute 'qualified_only'}
VAR_GLOBAL
	// Resultado esperado = 198
	iResultado_POU_CFC : INT;
	// Resultado esperado = 112	
	iResultado_POU_FBD : INT;
	// Resultado esperado = 118
	iResultado_POU_IL : INT;
	// Resultado esperado = 112
	iResultado_POU_LD : INT;
	// Resultado esperado = true
	bResultado_POU_SFC : BOOL;
END_VAR

// Device/Application/UserGVLs/Redundant/PIDs
{attribute 'qualified_only'}
VAR_GLOBAL
	// Set Point
	rPID_SP : REAL := 15000;
	// Preset Value
	rPID_PV : REAL;
	// Manipulated Variable
	rPID_MV : REAL;
END_VAR

